LIN {X 0,Y 179.067,Z 302.942,A -85,B 0,C 180,E1 -23619.497,E2 -23619.497} C_VEL
LIN {X 0,Y 181.423,Z 310.34,A -85,B 0,C 180,E1 -23622.061,E2 -23622.061} C_VEL
LIN {X 0,Y 182.867,Z 318.039,A -85,B 0,C 180,E1 -23624.448,E2 -23624.448} C_VEL
LIN {X 0,Y 183.604,Z 326.943,A -85,B 0,C 180,E1 -23627.105,E2 -23627.105} C_VEL
LIN {X 0,Y 183.542,Z 336.442,A -85,B 0,C 180,E1 -23629.98,E2 -23629.98} C_VEL
LIN {X 0,Y 183.368,Z 338.748,A -85,B 0,C 180,E1 -23630.712,E2 -23630.712} C_VEL
LIN {X 0,Y 178.856,Z 348.683,A -85,B 0,C 180,E1 -23633.185,E2 -23633.185} C_VEL
LIN {X 0,Y 173.994,Z 358.418,A -85,B 0,C 180,E1 -23636.262,E2 -23636.262} C_VEL
LIN {X 0,Y 169.557,Z 366.492,A -85,B 0,C 180,E1 -23639.486,E2 -23639.486} C_VEL
LIN {X 0,Y 165.463,Z 373.643,A -85,B 0,C 180,E1 -23643.123,E2 -23643.123} C_VEL
LIN {X 0,Y 162.202,Z 379.606,A -85,B 0,C 180,E1 -23647.048,E2 -23647.048} C_VEL
LIN {X 0,Y 158.721,Z 385.275,A -85,B 0,C 180,E1 -23651.944,E2 -23651.944} C_VEL
LIN {X 0,Y 156.544,Z 389.385,A -85,B 0,C 180,E1 -23657.028,E2 -23657.028} C_VEL
LIN {X 0,Y 155.24,Z 392.068,A -85,B 0,C 180,E1 -23662.194,E2 -23662.194} C_VEL
LIN {X 0,Y 154.776,Z 393.405,A -85,B 0,C 180,E1 -23667.398,E2 -23667.398} C_VEL
LIN {X 0,Y 154.745,Z 393.581,A -85,B 0,C 180,E1 -23670,E2 -23670} C_VEL
LIN {X 0,Y 154.935,Z 392.95,A -85,B 0,C 180,E1 -23675.205,E2 -23675.205} C_VEL
LIN {X 0,Y 155.776,Z 390.989,A -85,B 0,C 180,E1 -23680.397,E2 -23680.397} C_VEL
LIN {X 0,Y 157.497,Z 387.65,A -85,B 0,C 180,E1 -23685.53,E2 -23685.53} C_VEL
LIN {X 0,Y 159.441,Z 384.203,A -85,B 0,C 180,E1 -23689.305,E2 -23689.305} C_VEL
LIN {X 0,Y 162.138,Z 379.816,A -85,B 0,C 180,E1 -23692.962,E2 -23692.962} C_VEL
LIN {X 0,Y 165.058,Z 374.417,A -85,B 0,C 180,E1 -23696.599,E2 -23696.599} C_VEL
LIN {X 0,Y 169.475,Z 366.809,A -85,B 0,C 180,E1 -23700.531,E2 -23700.531} C_VEL
LIN {X 0,Y 173.917,Z 358.8,A -85,B 0,C 180,E1 -23703.755,E2 -23703.755} C_VEL
LIN {X 0,Y 178.733,Z 349.14,A -85,B 0,C 180,E1 -23706.845,E2 -23706.845} C_VEL
LIN {X 0,Y 183.37,Z 339.114,A -85,B 0,C 180,E1 -23709.349,E2 -23709.349} C_VEL
LIN {X 0,Y 183.799,Z 330.673,A -85,B 0,C 180,E1 -23711.941,E2 -23711.941} C_VEL
LIN {X 0,Y 183.309,Z 320.833,A -85,B 0,C 180,E1 -23714.875,E2 -23714.875} C_VEL
LIN {X 0,Y 181.97,Z 312.358,A -85,B 0,C 180,E1 -23717.475,E2 -23717.475} C_VEL
LIN {X 0,Y 179.973,Z 305.35,A -85,B 0,C 180,E1 -23719.831,E2 -23719.831} C_VEL
LIN {X 0,Y 177.108,Z 298.214,A -85,B 0,C 180,E1 -23722.528,E2 -23722.528} C_VEL
LIN {X 0,Y 174.424,Z 292.131,A -85,B 0,C 180,E1 -23724.958,E2 -23724.958} C_VEL
LIN {X 0,Y 171.473,Z 286.759,A -85,B 0,C 180,E1 -23727.456,E2 -23727.456} C_VEL
LIN {X 0,Y 168.98,Z 282.347,A -85,B 0,C 180,E1 -23729.657,E2 -23729.657} C_VEL
LIN {X 0,Y 166.592,Z 279.117,A -85,B 0,C 180,E1 -23731.666,E2 -23731.666} C_VEL
LIN {X 0,Y 165.823,Z 277.609,A -85,B 0,C 180,E1 -23732.439,E2 -23732.439} C_VEL
LIN {X 0,Y 163.535,Z 275.533,A -85,B 0,C 180,E1 -23734.403,E2 -23734.403} C_VEL
LIN {X 0,Y 162.075,Z 272.586,A -85,B 0,C 180,E1 -23736.004,E2 -23736.004} C_VEL
LIN {X 0,Y 158.994,Z 270.202,A -85,B 0,C 180,E1 -23739.121,E2 -23739.121} C_VEL
LIN {X 0,Y 157.602,Z 267.461,A -85,B 0,C 180,E1 -23740.958,E2 -23740.958} C_VEL
LIN {X 0,Y 157.402,Z 266.502,A -85,B 0,C 180,E1 -23741.446,E2 -23741.446} C_VEL
LIN {X 0,Y 157.532,Z 266.485,A -85,B 0,C 180,E1 -23747.111,E2 -23747.111} C_VEL
LIN {X 0,Y 157.691,Z 266.465,A -85,B 0,C 180,E1 -23749.731,E2 -23749.731} C_VEL
LIN {X 0,Y 157.768,Z 266.455,A -85,B 0,C 180,E1 -23752.32,E2 -23752.32} C_VEL
LIN {X 0,Y 158.247,Z 266.395,A -85,B 0,C 180,E1 -23760,E2 -23760} C_VEL
LIN {X 0,Y 157.764,Z 266.456,A -85,B 0,C 180,E1 -23767.68,E2 -23767.68} C_VEL
LIN {X 0,Y 157.635,Z 266.476,A -85,B 0,C 180,E1 -23771.228,E2 -23771.228} C_VEL
LIN {X 0,Y 157.436,Z 266.501,A -85,B 0,C 180,E1 -23775.536,E2 -23775.536} C_VEL
LIN {X 0,Y 157.532,Z 267.283,A -85,B 0,C 180,E1 -23778.666,E2 -23778.666} C_VEL
LIN {X 0,Y 158.727,Z 270.174,A -85,B 0,C 180,E1 -23780.334,E2 -23780.334} C_VEL
LIN {X 0,Y 161.142,Z 273.06,A -85,B 0,C 180,E1 -23782.942,E2 -23782.942} C_VEL
LIN {X 0,Y 162.364,Z 274.144,A -85,B 0,C 180,E1 -23784.111,E2 -23784.111} C_VEL
LIN {X 0,Y 164.013,Z 277.665,A -85,B 0,C 180,E1 -23785.9,E2 -23785.9} C_VEL
LIN {X 0,Y 166.386,Z 280.501,A -85,B 0,C 180,E1 -23787.967,E2 -23787.967} C_VEL
LIN {X 0,Y 168.328,Z 284.343,A -85,B 0,C 180,E1 -23789.809,E2 -23789.809} C_VEL
LIN {X 0,Y 169.782,Z 286.384,A -85,B 0,C 180,E1 -23790.977,E2 -23790.977} C_VEL
LIN {X 0,Y 172.139,Z 290.716,A -85,B 0,C 180,E1 -23793.01,E2 -23793.01} C_VEL
LIN {X 0,Y 176.395,Z 299.815,A -85,B 0,C 180,E1 -23796.701,E2 -23796.701} C_VEL
LIN {X 0,Y 179.977,Z 309.787,A -85,B 0,C 180,E1 -23800.222,E2 -23800.222} C_VEL
LIN {X 0,Y 181.352,Z 315.544,A -85,B 0,C 180,E1 -23802.016,E2 -23802.016} C_VEL
LIN {X 0,Y 182.317,Z 324.212,A -85,B 0,C 180,E1 -23804.451,E2 -23804.451} C_VEL
LIN {X 0,Y 182.511,Z 333.34,A -85,B 0,C 180,E1 -23807.024,E2 -23807.024} C_VEL
LIN {X 0,Y 181.857,Z 342.337,A -85,B 0,C 180,E1 -23809.595,E2 -23809.595} C_VEL
LIN {X 0,Y 181.369,Z 346.338,A -85,B 0,C 180,E1 -23810.804,E2 -23810.804} C_VEL
LIN {X 0,Y 178.739,Z 352.649,A -85,B 0,C 180,E1 -23812.449,E2 -23812.449} C_VEL
LIN {X 0,Y 173.678,Z 362.679,A -85,B 0,C 180,E1 -23815.492,E2 -23815.492} C_VEL
LIN {X 0,Y 169.218,Z 371.013,A -85,B 0,C 180,E1 -23818.724,E2 -23818.724} C_VEL
LIN {X 0,Y 164.754,Z 378.985,A -85,B 0,C 180,E1 -23822.705,E2 -23822.705} C_VEL
LIN {X 0,Y 161.215,Z 385.41,A -85,B 0,C 180,E1 -23826.899,E2 -23826.899} C_VEL
LIN {X 0,Y 158.016,Z 391.107,A -85,B 0,C 180,E1 -23831.86,E2 -23831.86} C_VEL
LIN {X 0,Y 155.897,Z 395.243,A -85,B 0,C 180,E1 -23836.973,E2 -23836.973} C_VEL
LIN {X 0,Y 154.871,Z 397.949,A -85,B 0,C 180,E1 -23842.175,E2 -23842.175} C_VEL
LIN {X 0,Y 154.685,Z 398.789,A -85,B 0,C 180,E1 -23844.786,E2 -23844.786} C_VEL
LIN {X 0,Y 154.744,Z 399.455,A -85,B 0,C 180,E1 -23850,E2 -23850} C_VEL
LIN {X 0,Y 154.683,Z 398.767,A -85,B 0,C 180,E1 -23855.213,E2 -23855.213} C_VEL
LIN {X 0,Y 155.277,Z 396.729,A -85,B 0,C 180,E1 -23860.43,E2 -23860.43} C_VEL
LIN {X 0,Y 156.762,Z 393.297,A -85,B 0,C 180,E1 -23865.604,E2 -23865.604} C_VEL
LIN {X 0,Y 159.448,Z 388.372,A -85,B 0,C 180,E1 -23870.647,E2 -23870.647} C_VEL
LIN {X 0,Y 162.167,Z 383.399,A -85,B 0,C 180,E1 -23874.481,E2 -23874.481} C_VEL
LIN {X 0,Y 165.93,Z 376.75,A -85,B 0,C 180,E1 -23878.457,E2 -23878.457} C_VEL
LIN {X 0,Y 167.766,Z 373.489,A -85,B 0,C 180,E1 -23880.084,E2 -23880.084} C_VEL
LIN {X 0,Y 169.015,Z 370.186,A -85,B 0,C 180,E1 -23881.698,E2 -23881.698} C_VEL
LIN {X 0,Y 169.665,Z 364.547,A -85,B 0,C 180,E1 -23884.452,E2 -23884.452} C_VEL
LIN {X 0,Y 170.538,Z 358.436,A -85,B 0,C 180,E1 -23887.058,E2 -23887.058} C_VEL
LIN {X 0,Y 172.074,Z 354.374,A -85,B 0,C 180,E1 -23888.397,E2 -23888.397} C_VEL
LIN {X 0,Y 174.942,Z 348.416,A -85,B 0,C 180,E1 -23889.999,E2 -23889.999} C_VEL
LIN {X 0,Y 176.332,Z 338.706,A -85,B 0,C 180,E1 -23893.011,E2 -23893.011} C_VEL
LIN {X 0,Y 176.669,Z 328.607,A -85,B 0,C 180,E1 -23896.035,E2 -23896.035} C_VEL
LIN {X 0,Y 176.019,Z 319.46,A -85,B 0,C 180,E1 -23898.793,E2 -23898.793} C_VEL
LIN {X 0,Y 174.653,Z 312.885,A -85,B 0,C 180,E1 -23900.986,E2 -23900.986} C_VEL
LIN {X 0,Y 171.698,Z 304.092,A -85,B 0,C 180,E1 -23904.318,E2 -23904.318} C_VEL
LIN {X 0,Y 168.228,Z 295.98,A -85,B 0,C 180,E1 -23907.815,E2 -23907.815} C_VEL
LIN {X 0,Y 165.717,Z 291.022,A -85,B 0,C 180,E1 -23910.287,E2 -23910.287} C_VEL
LIN {X 0,Y 163.651,Z 287.391,A -85,B 0,C 180,E1 -23912.332,E2 -23912.332} C_VEL
LIN {X 0,Y 163.002,Z 285.935,A -85,B 0,C 180,E1 -23913.082,E2 -23913.082} C_VEL
LIN {X 0,Y 160.702,Z 282.751,A -85,B 0,C 180,E1 -23915.371,E2 -23915.371} C_VEL
LIN {X 0,Y 159.58,Z 280.103,A -85,B 0,C 180,E1 -23916.821,E2 -23916.821} C_VEL
LIN {X 0,Y 156.897,Z 277.104,A -85,B 0,C 180,E1 -23919.849,E2 -23919.849} C_VEL
LIN {X 0,Y 155.347,Z 273.679,A -85,B 0,C 180,E1 -23922.22,E2 -23922.22} C_VEL
LIN {X 0,Y 151.929,Z 270.812,A -85,B 0,C 180,E1 -23927.587,E2 -23927.587} C_VEL
LIN {X 0,Y 150.752,Z 267.956,A -85,B 0,C 180,E1 -23930.694,E2 -23930.694} C_VEL
LIN {X 0,Y 150.654,Z 267.344,A -85,B 0,C 180,E1 -23931.28,E2 -23931.28} C_VEL
LIN {X 0,Y 150.892,Z 267.312,A -85,B 0,C 180,E1 -23937.331,E2 -23937.331} C_VEL
LIN {X 0,Y 151.215,Z 267.273,A -85,B 0,C 180,E1 -23940,E2 -23940} C_VEL
LIN {X 0,Y 150.706,Z 267.338,A -85,B 0,C 180,E1 -23948.042,E2 -23948.042} C_VEL
LIN {X 0,Y 150.671,Z 267.462,A -85,B 0,C 180,E1 -23949.312,E2 -23949.312} C_VEL
LIN {X 0,Y 151.617,Z 270.359,A -85,B 0,C 180,E1 -23952.124,E2 -23952.124} C_VEL
LIN {X 0,Y 153.898,Z 272.667,A -85,B 0,C 180,E1 -23956.243,E2 -23956.243} C_VEL
LIN {X 0,Y 155.476,Z 273.555,A -85,B 0,C 180,E1 -23958.363,E2 -23958.363} C_VEL
LIN {X 0,Y 156.748,Z 276.518,A -85,B 0,C 180,E1 -23960.35,E2 -23960.35} C_VEL
LIN {X 0,Y 159.096,Z 278.658,A -85,B 0,C 180,E1 -23963.021,E2 -23963.021} C_VEL
LIN {X 0,Y 159.656,Z 279.316,A -85,B 0,C 180,E1 -23963.64,E2 -23963.64} C_VEL
LIN {X 0,Y 161.407,Z 282.44,A -85,B 0,C 180,E1 -23965.668,E2 -23965.668} C_VEL
LIN {X 0,Y 163.234,Z 284.363,A -85,B 0,C 180,E1 -23967.397,E2 -23967.397} C_VEL
LIN {X 0,Y 165.077,Z 287.673,A -85,B 0,C 180,E1 -23969.315,E2 -23969.315} C_VEL
LIN {X 0,Y 166.892,Z 290.685,A -85,B 0,C 180,E1 -23971.055,E2 -23971.055} C_VEL
LIN {X 0,Y 168.682,Z 294.057,A -85,B 0,C 180,E1 -23972.795,E2 -23972.795} C_VEL
LIN {X 0,Y 171.593,Z 300.422,A -85,B 0,C 180,E1 -23975.707,E2 -23975.707} C_VEL
LIN {X 0,Y 174.378,Z 307.594,A -85,B 0,C 180,E1 -23978.661,E2 -23978.661} C_VEL
LIN {X 0,Y 176.279,Z 314.277,A -85,B 0,C 180,E1 -23981.134,E2 -23981.134} C_VEL
LIN {X 0,Y 177.396,Z 321.698,A -85,B 0,C 180,E1 -23983.604,E2 -23983.604} C_VEL
LIN {X 0,Y 177.79,Z 330.811,A -85,B 0,C 180,E1 -23986.487,E2 -23986.487} C_VEL
LIN {X 0,Y 177.353,Z 340.066,A -85,B 0,C 180,E1 -23989.516,E2 -23989.516} C_VEL
LIN {X 0,Y 172.297,Z 350.598,A -85,B 0,C 180,E1 -23992.277,E2 -23992.277} C_VEL
LIN {X 0,Y 167.318,Z 360.036,A -85,B 0,C 180,E1 -23995.455,E2 -23995.455} C_VEL
LIN {X 0,Y 162.038,Z 369.033,A -85,B 0,C 180,E1 -23999.361,E2 -23999.361} C_VEL
LIN {X 0,Y 157.689,Z 376.278,A -85,B 0,C 180,E1 -24003.533,E2 -24003.533} C_VEL
LIN {X 0,Y 154.631,Z 381.346,A -85,B 0,C 180,E1 -24007.274,E2 -24007.274} C_VEL
LIN {X 0,Y 151.296,Z 386.595,A -85,B 0,C 180,E1 -24012.426,E2 -24012.426} C_VEL
LIN {X 0,Y 149.628,Z 389.521,A -85,B 0,C 180,E1 -24016.418,E2 -24016.418} C_VEL
LIN {X 0,Y 148.211,Z 392.204,A -85,B 0,C 180,E1 -24021.822,E2 -24021.822} C_VEL
LIN {X 0,Y 147.68,Z 393.54,A -85,B 0,C 180,E1 -24027.273,E2 -24027.273} C_VEL
LIN {X 0,Y 147.631,Z 393.649,A -85,B 0,C 180,E1 -24031.363,E2 -24031.363} C_VEL
LIN {X 0,Y 147.861,Z 393.084,A -85,B 0,C 180,E1 -24035.455,E2 -24035.455} C_VEL
LIN {X 0,Y 148.777,Z 391.124,A -85,B 0,C 180,E1 -24040.892,E2 -24040.892} C_VEL
LIN {X 0,Y 150.649,Z 387.785,A -85,B 0,C 180,E1 -24046.255,E2 -24046.255} C_VEL
LIN {X 0,Y 152.738,Z 384.337,A -85,B 0,C 180,E1 -24050.188,E2 -24050.188} C_VEL
LIN {X 0,Y 155.581,Z 379.951,A -85,B 0,C 180,E1 -24053.989,E2 -24053.989} C_VEL
LIN {X 0,Y 158.893,Z 374.274,A -85,B 0,C 180,E1 -24057.915,E2 -24057.915} C_VEL
LIN {X 0,Y 163.392,Z 366.942,A -85,B 0,C 180,E1 -24061.797,E2 -24061.797} C_VEL
LIN {X 0,Y 168.039,Z 358.933,A -85,B 0,C 180,E1 -24065.105,E2 -24065.105} C_VEL
LIN {X 0,Y 173.103,Z 349.272,A -85,B 0,C 180,E1 -24068.255,E2 -24068.255} C_VEL
LIN {X 0,Y 177.411,Z 340.434,A -85,B 0,C 180,E1 -24070.528,E2 -24070.528} C_VEL
LIN {X 0,Y 177.889,Z 332.538,A -85,B 0,C 180,E1 -24073.106,E2 -24073.106} C_VEL
LIN {X 0,Y 177.721,Z 324.154,A -85,B 0,C 180,E1 -24075.775,E2 -24075.775} C_VEL
LIN {X 0,Y 176.688,Z 316.064,A -85,B 0,C 180,E1 -24078.431,E2 -24078.431} C_VEL
LIN {X 0,Y 175.206,Z 310.11,A -85,B 0,C 180,E1 -24080.573,E2 -24080.573} C_VEL
LIN {X 0,Y 172.379,Z 302.202,A -85,B 0,C 180,E1 -24083.759,E2 -24083.759} C_VEL
LIN {X 0,Y 168.362,Z 293.124,A -85,B 0,C 180,E1 -24087.844,E2 -24087.844} C_VEL
LIN {X 0,Y 165.703,Z 288.288,A -85,B 0,C 180,E1 -24090.458,E2 -24090.458} C_VEL
LIN {X 0,Y 163.476,Z 284.804,A -85,B 0,C 180,E1 -24092.647,E2 -24092.647} C_VEL
LIN {X 0,Y 162.93,Z 283.848,A -85,B 0,C 180,E1 -24093.242,E2 -24093.242} C_VEL
LIN {X 0,Y 160.632,Z 281.334,A -85,B 0,C 180,E1 -24095.487,E2 -24095.487} C_VEL
LIN {X 0,Y 159.396,Z 278.805,A -85,B 0,C 180,E1 -24097.049,E2 -24097.049} C_VEL
LIN {X 0,Y 157.027,Z 276.836,A -85,B 0,C 180,E1 -24099.705,E2 -24099.705} C_VEL
LIN {X 0,Y 155.571,Z 273.871,A -85,B 0,C 180,E1 -24101.906,E2 -24101.906} C_VEL
LIN {X 0,Y 155.406,Z 273.314,A -85,B 0,C 180,E1 -24102.226,E2 -24102.226} C_VEL
LIN {X 0,Y 152.481,Z 271.504,A -85,B 0,C 180,E1 -24106.676,E2 -24106.676} C_VEL
LIN {X 0,Y 150.953,Z 268.682,A -85,B 0,C 180,E1 -24110.453,E2 -24110.453} C_VEL
LIN {X 0,Y 150.692,Z 267.336,A -85,B 0,C 180,E1 -24111.788,E2 -24111.788} C_VEL
LIN {X 0,Y 151.209,Z 267.272,A -85,B 0,C 180,E1 -24120,E2 -24120} C_VEL
LIN {X 0,Y 150.719,Z 267.523,A -85,B 0,C 180,E1 -24128.294,E2 -24128.294} C_VEL
LIN {X 0,Y 151.32,Z 269.624,A -85,B 0,C 180,E1 -24130.368,E2 -24130.368} C_VEL
LIN {X 0,Y 153.209,Z 272.203,A -85,B 0,C 180,E1 -24134.274,E2 -24134.274} C_VEL
LIN {X 0,Y 155.638,Z 274.025,A -85,B 0,C 180,E1 -24137.831,E2 -24137.831} C_VEL
LIN {X 0,Y 157.461,Z 277.866,A -85,B 0,C 180,E1 -24140.544,E2 -24140.544} C_VEL
LIN {X 0,Y 159.847,Z 280.493,A -85,B 0,C 180,E1 -24143.224,E2 -24143.224} C_VEL
LIN {X 0,Y 161.591,Z 284.192,A -85,B 0,C 180,E1 -24145.349,E2 -24145.349} C_VEL
LIN {X 0,Y 163.459,Z 286.72,A -85,B 0,C 180,E1 -24147.182,E2 -24147.182} C_VEL
LIN {X 0,Y 165.243,Z 290.402,A -85,B 0,C 180,E1 -24149.107,E2 -24149.107} C_VEL
LIN {X 0,Y 166.06,Z 291.49,A -85,B 0,C 180,E1 -24149.82,E2 -24149.82} C_VEL
LIN {X 0,Y 168.947,Z 297.6,A -85,B 0,C 180,E1 -24152.737,E2 -24152.737} C_VEL
LIN {X 0,Y 172.405,Z 305.804,A -85,B 0,C 180,E1 -24156.234,E2 -24156.234} C_VEL
LIN {X 0,Y 174.848,Z 313.347,A -85,B 0,C 180,E1 -24159.08,E2 -24159.08} C_VEL
LIN {X 0,Y 176.143,Z 319.606,A -85,B 0,C 180,E1 -24161.172,E2 -24161.172} C_VEL
LIN {X 0,Y 176.759,Z 328.96,A -85,B 0,C 180,E1 -24163.984,E2 -24163.984} C_VEL
LIN {X 0,Y 176.519,Z 337.676,A -85,B 0,C 180,E1 -24166.601,E2 -24166.601} C_VEL
LIN {X 0,Y 175.31,Z 347.396,A -85,B 0,C 180,E1 -24169.613,E2 -24169.613} C_VEL
LIN {X 0,Y 174.02,Z 350.627,A -85,B 0,C 180,E1 -24170.499,E2 -24170.499} C_VEL
LIN {X 0,Y 168.732,Z 361.032,A -85,B 0,C 180,E1 -24173.591,E2 -24173.591} C_VEL
LIN {X 0,Y 163.915,Z 369.618,A -85,B 0,C 180,E1 -24176.861,E2 -24176.861} C_VEL
LIN {X 0,Y 159.05,Z 377.839,A -85,B 0,C 180,E1 -24180.918,E2 -24180.918} C_VEL
LIN {X 0,Y 155.539,Z 383.693,A -85,B 0,C 180,E1 -24184.648,E2 -24184.648} C_VEL
LIN {X 0,Y 152.791,Z 388.328,A -85,B 0,C 180,E1 -24188.409,E2 -24188.409} C_VEL
LIN {X 0,Y 149.896,Z 393.225,A -85,B 0,C 180,E1 -24193.661,E2 -24193.661} C_VEL
LIN {X 0,Y 148.272,Z 396.635,A -85,B 0,C 180,E1 -24199.07,E2 -24199.07} C_VEL
LIN {X 0,Y 147.612,Z 398.654,A -85,B 0,C 180,E1 -24204.536,E2 -24204.536} C_VEL
LIN {X 0,Y 147.656,Z 399.32,A -85,B 0,C 180,E1 -24210,E2 -24210} C_VEL
LIN {X 0,Y 147.61,Z 398.632,A -85,B 0,C 180,E1 -24215.464,E2 -24215.464} C_VEL
LIN {X 0,Y 148.271,Z 396.594,A -85,B 0,C 180,E1 -24220.929,E2 -24220.929} C_VEL
LIN {X 0,Y 149.892,Z 393.16,A -85,B 0,C 180,E1 -24226.339,E2 -24226.339} C_VEL
LIN {X 0,Y 152.778,Z 388.235,A -85,B 0,C 180,E1 -24231.593,E2 -24231.593} C_VEL
LIN {X 0,Y 156.652,Z 381.67,A -85,B 0,C 180,E1 -24236.656,E2 -24236.656} C_VEL
LIN {X 0,Y 161.019,Z 374.371,A -85,B 0,C 180,E1 -24240.854,E2 -24240.854} C_VEL
LIN {X 0,Y 166.195,Z 365.331,A -85,B 0,C 180,E1 -24244.812,E2 -24244.812} C_VEL
LIN {X 0,Y 171.334,Z 355.855,A -85,B 0,C 180,E1 -24247.973,E2 -24247.973} C_VEL
LIN {X 0,Y 172.074,Z 354.374,A -85,B 0,C 180,E1 -24248.397,E2 -24248.397} C_VEL
LIN {X 0,Y 173.06,Z 351.66,A -85,B 0,C 180,E1 -24249.261,E2 -24249.261} C_VEL
LIN {X 0,Y 173.329,Z 347.715,A -85,B 0,C 180,E1 -24250.724,E2 -24250.724} C_VEL
LIN {X 0,Y 172.71,Z 344.045,A -85,B 0,C 180,E1 -24252.275,E2 -24252.275} C_VEL
LIN {X 0,Y 171.017,Z 336.395,A -85,B 0,C 180,E1 -24255.458,E2 -24255.458} C_VEL
LIN {X 0,Y 170.946,Z 333.508,A -85,B 0,C 180,E1 -24256.433,E2 -24256.433} C_VEL
LIN {X 0,Y 170.857,Z 324.847,A -85,B 0,C 180,E1 -24259.204,E2 -24259.204} C_VEL
LIN {X 0,Y 169.871,Z 317.824,A -85,B 0,C 180,E1 -24261.641,E2 -24261.641} C_VEL
LIN {X 0,Y 167.569,Z 309.915,A -85,B 0,C 180,E1 -24264.809,E2 -24264.809} C_VEL
LIN {X 0,Y 164.492,Z 301.734,A -85,B 0,C 180,E1 -24268.513,E2 -24268.513} C_VEL
LIN {X 0,Y 162.458,Z 297.122,A -85,B 0,C 180,E1 -24270.878,E2 -24270.878} C_VEL
LIN {X 0,Y 159.428,Z 291.4,A -85,B 0,C 180,E1 -24274.37,E2 -24274.37} C_VEL
LIN {X 0,Y 157.388,Z 287.639,A -85,B 0,C 180,E1 -24276.914,E2 -24276.914} C_VEL
LIN {X 0,Y 156.806,Z 286.281,A -85,B 0,C 180,E1 -24277.78,E2 -24277.78} C_VEL
LIN {X 0,Y 154.507,Z 283.311,A -85,B 0,C 180,E1 -24280.75,E2 -24280.75} C_VEL
LIN {X 0,Y 153.427,Z 280.414,A -85,B 0,C 180,E1 -24282.764,E2 -24282.764} C_VEL
LIN {X 0,Y 150.236,Z 277.448,A -85,B 0,C 180,E1 -24288.331,E2 -24288.331} C_VEL
LIN {X 0,Y 149.201,Z 274.279,A -85,B 0,C 180,E1 -24291.876,E2 -24291.876} C_VEL
LIN {X 0,Y 147.773,Z 273.479,A -85,B 0,C 180,E1 -24300,E2 -24300} C_VEL
LIN {X 0,Y 149.213,Z 274.312,A -85,B 0,C 180,E1 -24308.635,E2 -24308.635} C_VEL
LIN {X 0,Y 150.133,Z 277.31,A -85,B 0,C 180,E1 -24311.912,E2 -24311.912} C_VEL
LIN {X 0,Y 152.264,Z 279.562,A -85,B 0,C 180,E1 -24316.078,E2 -24316.078} C_VEL
LIN {X 0,Y 153.329,Z 280.245,A -85,B 0,C 180,E1 -24317.636,E2 -24317.636} C_VEL
LIN {X 0,Y 154.634,Z 283.227,A -85,B 0,C 180,E1 -24319.93,E2 -24319.93} C_VEL
LIN {X 0,Y 156.999,Z 285.641,A -85,B 0,C 180,E1 -24322.886,E2 -24322.886} C_VEL
LIN {X 0,Y 158.503,Z 288.594,A -85,B 0,C 180,E1 -24324.912,E2 -24324.912} C_VEL
LIN {X 0,Y 159.669,Z 289.817,A -85,B 0,C 180,E1 -24326.114,E2 -24326.114} C_VEL
LIN {X 0,Y 162.989,Z 295.615,A -85,B 0,C 180,E1 -24329.87,E2 -24329.87} C_VEL
LIN {X 0,Y 166.061,Z 302.275,A -85,B 0,C 180,E1 -24333.38,E2 -24333.38} C_VEL
LIN {X 0,Y 169.043,Z 310.375,A -85,B 0,C 180,E1 -24337.075,E2 -24337.075} C_VEL
LIN {X 0,Y 171.126,Z 318.459,A -85,B 0,C 180,E1 -24340.304,E2 -24340.304} C_VEL
LIN {X 0,Y 171.991,Z 326.656,A -85,B 0,C 180,E1 -24343.193,E2 -24343.193} C_VEL
LIN {X 0,Y 171.835,Z 336.017,A -85,B 0,C 180,E1 -24346.356,E2 -24346.356} C_VEL
LIN {X 0,Y 171.376,Z 341.47,A -85,B 0,C 180,E1 -24348.257,E2 -24348.257} C_VEL
LIN {X 0,Y 165.839,Z 352.438,A -85,B 0,C 180,E1 -24351.312,E2 -24351.312} C_VEL
LIN {X 0,Y 160.684,Z 361.565,A -85,B 0,C 180,E1 -24354.583,E2 -24354.583} C_VEL
LIN {X 0,Y 155.229,Z 370.282,A -85,B 0,C 180,E1 -24358.624,E2 -24358.624} C_VEL
LIN {X 0,Y 151.343,Z 376.414,A -85,B 0,C 180,E1 -24362.33,E2 -24362.33} C_VEL
LIN {X 0,Y 148.092,Z 381.482,A -85,B 0,C 180,E1 -24366.21,E2 -24366.21} C_VEL
LIN {X 0,Y 144.512,Z 386.731,A -85,B 0,C 180,E1 -24371.572,E2 -24371.572} C_VEL
LIN {X 0,Y 142.708,Z 389.657,A -85,B 0,C 180,E1 -24375.745,E2 -24375.745} C_VEL
LIN {X 0,Y 141.165,Z 392.339,A -85,B 0,C 180,E1 -24381.411,E2 -24381.411} C_VEL
LIN {X 0,Y 140.594,Z 393.675,A -85,B 0,C 180,E1 -24387.135,E2 -24387.135} C_VEL
LIN {X 0,Y 140.561,Z 393.85,A -85,B 0,C 180,E1 -24390,E2 -24390} C_VEL
LIN {X 0,Y 140.799,Z 393.219,A -85,B 0,C 180,E1 -24395.73,E2 -24395.73} C_VEL
LIN {X 0,Y 141.802,Z 391.258,A -85,B 0,C 180,E1 -24401.435,E2 -24401.435} C_VEL
LIN {X 0,Y 143.81,Z 387.919,A -85,B 0,C 180,E1 -24407.051,E2 -24407.051} C_VEL
LIN {X 0,Y 146.077,Z 384.471,A -85,B 0,C 180,E1 -24411.152,E2 -24411.152} C_VEL
LIN {X 0,Y 149.064,Z 380.085,A -85,B 0,C 180,E1 -24415.108,E2 -24415.108} C_VEL
LIN {X 0,Y 152.837,Z 374.089,A -85,B 0,C 180,E1 -24419.365,E2 -24419.365} C_VEL
LIN {X 0,Y 158.174,Z 365.848,A -85,B 0,C 180,E1 -24423.739,E2 -24423.739} C_VEL
LIN {X 0,Y 163.13,Z 357.585,A -85,B 0,C 180,E1 -24427.096,E2 -24427.096} C_VEL
LIN {X 0,Y 168.517,Z 347.628,A -85,B 0,C 180,E1 -24430.273,E2 -24430.273} C_VEL
LIN {X 0,Y 171.488,Z 341.782,A -85,B 0,C 180,E1 -24431.788,E2 -24431.788} C_VEL
LIN {X 0,Y 172.12,Z 332.707,A -85,B 0,C 180,E1 -24434.924,E2 -24434.924} C_VEL
LIN {X 0,Y 171.903,Z 323.637,A -85,B 0,C 180,E1 -24438.014,E2 -24438.014} C_VEL
LIN {X 0,Y 170.938,Z 317.042,A -85,B 0,C 180,E1 -24440.411,E2 -24440.411} C_VEL
LIN {X 0,Y 168.729,Z 309.394,A -85,B 0,C 180,E1 -24443.59,E2 -24443.59} C_VEL
LIN {X 0,Y 165.721,Z 301.506,A -85,B 0,C 180,E1 -24447.269,E2 -24447.269} C_VEL
LIN {X 0,Y 164.145,Z 297.962,A -85,B 0,C 180,E1 -24449.083,E2 -24449.083} C_VEL
LIN {X 0,Y 162.622,Z 294.578,A -85,B 0,C 180,E1 -24450.909,E2 -24450.909} C_VEL
LIN {X 0,Y 159.942,Z 290.097,A -85,B 0,C 180,E1 -24453.934,E2 -24453.934} C_VEL
LIN {X 0,Y 157.649,Z 287.113,A -85,B 0,C 180,E1 -24456.519,E2 -24456.519} C_VEL
LIN {X 0,Y 156.934,Z 285.349,A -85,B 0,C 180,E1 -24457.625,E2 -24457.625} C_VEL
LIN {X 0,Y 154.693,Z 283.245,A -85,B 0,C 180,E1 -24460.427,E2 -24460.427} C_VEL
LIN {X 0,Y 153.256,Z 280.015,A -85,B 0,C 180,E1 -24463.001,E2 -24463.001} C_VEL
LIN {X 0,Y 150.609,Z 278.032,A -85,B 0,C 180,E1 -24467.586,E2 -24467.586} C_VEL
LIN {X 0,Y 149.326,Z 274.871,A -85,B 0,C 180,E1 -24471.73,E2 -24471.73} C_VEL
LIN {X 0,Y 149.152,Z 274.273,A -85,B 0,C 180,E1 -24472.555,E2 -24472.555} C_VEL
LIN {X 0,Y 148.078,Z 273.648,A -85,B 0,C 180,E1 -24480,E2 -24480} C_VEL
LIN {X 0,Y 149.308,Z 274.423,A -85,B 0,C 180,E1 -24487.607,E2 -24487.607} C_VEL
LIN {X 0,Y 150.395,Z 277.626,A -85,B 0,C 180,E1 -24491.435,E2 -24491.435} C_VEL
LIN {X 0,Y 153.566,Z 280.712,A -85,B 0,C 180,E1 -24497.113,E2 -24497.113} C_VEL
LIN {X 0,Y 155.445,Z 284.749,A -85,B 0,C 180,E1 -24500.252,E2 -24500.252} C_VEL
LIN {X 0,Y 157.183,Z 286.833,A -85,B 0,C 180,E1 -24502.423,E2 -24502.423} C_VEL
LIN {X 0,Y 158.929,Z 290.681,A -85,B 0,C 180,E1 -24504.841,E2 -24504.841} C_VEL
LIN {X 0,Y 160.077,Z 292.12,A -85,B 0,C 180,E1 -24506.042,E2 -24506.042} C_VEL
LIN {X 0,Y 162.034,Z 296.489,A -85,B 0,C 180,E1 -24508.497,E2 -24508.497} C_VEL
LIN {X 0,Y 164.531,Z 301.686,A -85,B 0,C 180,E1 -24511.316,E2 -24511.316} C_VEL
LIN {X 0,Y 167.86,Z 310.54,A -85,B 0,C 180,E1 -24515.337,E2 -24515.337} C_VEL
LIN {X 0,Y 169.991,Z 318.018,A -85,B 0,C 180,E1 -24518.327,E2 -24518.327} C_VEL
LIN {X 0,Y 170.877,Z 323.847,A -85,B 0,C 180,E1 -24520.374,E2 -24520.374} C_VEL
LIN {X 0,Y 171.063,Z 332.96,A -85,B 0,C 180,E1 -24523.311,E2 -24523.311} C_VEL
LIN {X 0,Y 170.35,Z 342.245,A -85,B 0,C 180,E1 -24526.288,E2 -24526.288} C_VEL
LIN {X 0,Y 169.288,Z 348.534,A -85,B 0,C 180,E1 -24528.375,E2 -24528.375} C_VEL
LIN {X 0,Y 167.55,Z 352.574,A -85,B 0,C 180,E1 -24529.53,E2 -24529.53} C_VEL
LIN {X 0,Y 162.142,Z 362.413,A -85,B 0,C 180,E1 -24532.639,E2 -24532.639} C_VEL
LIN {X 0,Y 157.201,Z 370.746,A -85,B 0,C 180,E1 -24536.024,E2 -24536.024} C_VEL
LIN {X 0,Y 152.185,Z 378.717,A -85,B 0,C 180,E1 -24540.235,E2 -24540.235} C_VEL
LIN {X 0,Y 148.135,Z 385.14,A -85,B 0,C 180,E1 -24544.723,E2 -24544.723} C_VEL
LIN {X 0,Y 144.511,Z 390.837,A -85,B 0,C 180,E1 -24550.096,E2 -24550.096} C_VEL
LIN {X 0,Y 142.02,Z 394.974,A -85,B 0,C 180,E1 -24555.674,E2 -24555.674} C_VEL
LIN {X 0,Y 140.772,Z 397.68,A -85,B 0,C 180,E1 -24561.386,E2 -24561.386} C_VEL
LIN {X 0,Y 140.533,Z 398.519,A -85,B 0,C 180,E1 -24564.259,E2 -24564.259} C_VEL
LIN {X 0,Y 140.56,Z 399.186,A -85,B 0,C 180,E1 -24570,E2 -24570} C_VEL
LIN {X 0,Y 140.532,Z 398.496,A -85,B 0,C 180,E1 -24575.74,E2 -24575.74} C_VEL
LIN {X 0,Y 141.258,Z 396.457,A -85,B 0,C 180,E1 -24581.479,E2 -24581.479} C_VEL
LIN {X 0,Y 143.051,Z 393.024,A -85,B 0,C 180,E1 -24587.144,E2 -24587.144} C_VEL
LIN {X 0,Y 146.159,Z 388.099,A -85,B 0,C 180,E1 -24592.624,E2 -24592.624} C_VEL
LIN {X 0,Y 149.275,Z 383.159,A -85,B 0,C 180,E1 -24596.728,E2 -24596.728} C_VEL
LIN {X 0,Y 153.514,Z 376.475,A -85,B 0,C 180,E1 -24601,E2 -24601} C_VEL
LIN {X 0,Y 158.732,Z 367.946,A -85,B 0,C 180,E1 -24605.141,E2 -24605.141} C_VEL
LIN {X 0,Y 163.919,Z 359.051,A -85,B 0,C 180,E1 -24608.439,E2 -24608.439} C_VEL
LIN {X 0,Y 168.698,Z 350.022,A -85,B 0,C 180,E1 -24611.092,E2 -24611.092} C_VEL
LIN {X 0,Y 169.923,Z 344.11,A -85,B 0,C 180,E1 -24613.034,E2 -24613.034} C_VEL
LIN {X 0,Y 170.809,Z 336.133,A -85,B 0,C 180,E1 -24615.616,E2 -24615.616} C_VEL
LIN {X 0,Y 170.946,Z 333.508,A -85,B 0,C 180,E1 -24616.433,E2 -24616.433} C_VEL
LIN {X 0,Y 170.808,Z 330.777,A -85,B 0,C 180,E1 -24617.38,E2 -24617.38} C_VEL
LIN {X 0,Y 170.131,Z 328.361,A -85,B 0,C 180,E1 -24618.403,E2 -24618.403} C_VEL
LIN {X 0,Y 167.929,Z 324.217,A -85,B 0,C 180,E1 -24620.584,E2 -24620.584} C_VEL
LIN {X 0,Y 164.205,Z 318.223,A -85,B 0,C 180,E1 -24624.035,E2 -24624.035} C_VEL
LIN {X 0,Y 163.342,Z 315.872,A -85,B 0,C 180,E1 -24625.156,E2 -24625.156} C_VEL
LIN {X 0,Y 160.654,Z 307.629,A -85,B 0,C 180,E1 -24629.085,E2 -24629.085} C_VEL
LIN {X 0,Y 158.324,Z 301.993,A -85,B 0,C 180,E1 -24632.22,E2 -24632.22} C_VEL
LIN {X 0,Y 156.551,Z 297.822,A -85,B 0,C 180,E1 -24634.756,E2 -24634.756} C_VEL
LIN {X 0,Y 154.687,Z 294.464,A -85,B 0,C 180,E1 -24637.283,E2 -24637.283} C_VEL
LIN {X 0,Y 153.959,Z 292.502,A -85,B 0,C 180,E1 -24638.581,E2 -24638.581} C_VEL
LIN {X 0,Y 151.827,Z 289.282,A -85,B 0,C 180,E1 -24641.793,E2 -24641.793} C_VEL
LIN {X 0,Y 151.118,Z 287.004,A -85,B 0,C 180,E1 -24643.45,E2 -24643.45} C_VEL
LIN {X 0,Y 148.276,Z 284.016,A -85,B 0,C 180,E1 -24649.071,E2 -24649.071} C_VEL
LIN {X 0,Y 147.501,Z 281.157,A -85,B 0,C 180,E1 -24652.471,E2 -24652.471} C_VEL
LIN {X 0,Y 146.31,Z 280.423,A -85,B 0,C 180,E1 -24660,E2 -24660} C_VEL
LIN {X 0,Y 147.508,Z 281.308,A -85,B 0,C 180,E1 -24668.218,E2 -24668.218} C_VEL
LIN {X 0,Y 148.285,Z 284.173,A -85,B 0,C 180,E1 -24671.621,E2 -24671.621} C_VEL
LIN {X 0,Y 150.536,Z 286.477,A -85,B 0,C 180,E1 -24676.268,E2 -24676.268} C_VEL
LIN {X 0,Y 151.036,Z 287.135,A -85,B 0,C 180,E1 -24677.169,E2 -24677.169} C_VEL
LIN {X 0,Y 151.859,Z 289.247,A -85,B 0,C 180,E1 -24678.903,E2 -24678.903} C_VEL
LIN {X 0,Y 153.608,Z 291.353,A -85,B 0,C 180,E1 -24681.471,E2 -24681.471} C_VEL
LIN {X 0,Y 156.361,Z 295.754,A -85,B 0,C 180,E1 -24685.278,E2 -24685.278} C_VEL
LIN {X 0,Y 159.245,Z 301.173,A -85,B 0,C 180,E1 -24689.043,E2 -24689.043} C_VEL
LIN {X 0,Y 162.045,Z 308.012,A -85,B 0,C 180,E1 -24692.829,E2 -24692.829} C_VEL
LIN {X 0,Y 164.574,Z 316.149,A -85,B 0,C 180,E1 -24696.717,E2 -24696.717} C_VEL
LIN {X 0,Y 165.928,Z 322.553,A -85,B 0,C 180,E1 -24699.445,E2 -24699.445} C_VEL
LIN {X 0,Y 166.371,Z 329.317,A -85,B 0,C 180,E1 -24701.986,E2 -24701.986} C_VEL
LIN {X 0,Y 166.085,Z 337.106,A -85,B 0,C 180,E1 -24704.794,E2 -24704.794} C_VEL
LIN {X 0,Y 165.259,Z 343.463,A -85,B 0,C 180,E1 -24707.123,E2 -24707.123} C_VEL
LIN {X 0,Y 159.416,Z 354.197,A -85,B 0,C 180,E1 -24710.265,E2 -24710.265} C_VEL
LIN {X 0,Y 154.107,Z 363.051,A -85,B 0,C 180,E1 -24713.64,E2 -24713.64} C_VEL
LIN {X 0,Y 148.428,Z 371.53,A -85,B 0,C 180,E1 -24717.813,E2 -24717.813} C_VEL
LIN {X 0,Y 143.835,Z 378.35,A -85,B 0,C 180,E1 -24722.343,E2 -24722.343} C_VEL
LIN {X 0,Y 140.516,Z 383.053,A -85,B 0,C 180,E1 -24726.414,E2 -24726.414} C_VEL
LIN {X 0,Y 137.771,Z 386.867,A -85,B 0,C 180,E1 -24730.636,E2 -24730.636} C_VEL
LIN {X 0,Y 135.82,Z 389.793,A -85,B 0,C 180,E1 -24735.006,E2 -24735.006} C_VEL
LIN {X 0,Y 134.134,Z 392.475,A -85,B 0,C 180,E1 -24740.957,E2 -24740.957} C_VEL
LIN {X 0,Y 133.519,Z 393.81,A -85,B 0,C 180,E1 -24746.983,E2 -24746.983} C_VEL
LIN {X 0,Y 133.475,Z 393.985,A -85,B 0,C 180,E1 -24750,E2 -24750} C_VEL
LIN {X 0,Y 133.731,Z 393.353,A -85,B 0,C 180,E1 -24756.034,E2 -24756.034} C_VEL
LIN {X 0,Y 134.827,Z 391.393,A -85,B 0,C 180,E1 -24762.035,E2 -24762.035} C_VEL
LIN {X 0,Y 137.013,Z 388.054,A -85,B 0,C 180,E1 -24767.925,E2 -24767.925} C_VEL
LIN {X 0,Y 139.465,Z 384.605,A -85,B 0,C 180,E1 -24772.207,E2 -24772.207} C_VEL
LIN {X 0,Y 142.612,Z 380.22,A -85,B 0,C 180,E1 -24776.329,E2 -24776.329} C_VEL
LIN {X 0,Y 146.916,Z 373.878,A -85,B 0,C 180,E1 -24780.947,E2 -24780.947} C_VEL
LIN {X 0,Y 152.312,Z 365.981,A -85,B 0,C 180,E1 -24785.225,E2 -24785.225} C_VEL
LIN {X 0,Y 157.514,Z 357.717,A -85,B 0,C 180,E1 -24788.657,E2 -24788.657} C_VEL
LIN {X 0,Y 163.17,Z 347.759,A -85,B 0,C 180,E1 -24791.883,E2 -24791.883} C_VEL
LIN {X 0,Y 165.574,Z 343.094,A -85,B 0,C 180,E1 -24793.141,E2 -24793.141} C_VEL
LIN {X 0,Y 166.394,Z 334.354,A -85,B 0,C 180,E1 -24796.356,E2 -24796.356} C_VEL
LIN {X 0,Y 166.423,Z 326.815,A -85,B 0,C 180,E1 -24799.115,E2 -24799.115} C_VEL
LIN {X 0,Y 165.477,Z 319.613,A -85,B 0,C 180,E1 -24801.987,E2 -24801.987} C_VEL
LIN {X 0,Y 163.551,Z 312.47,A -85,B 0,C 180,E1 -24805.214,E2 -24805.214} C_VEL
LIN {X 0,Y 161.037,Z 305.378,A -85,B 0,C 180,E1 -24808.82,E2 -24808.82} C_VEL
LIN {X 0,Y 158.809,Z 300.046,A -85,B 0,C 180,E1 -24811.891,E2 -24811.891} C_VEL
LIN {X 0,Y 156.63,Z 296.029,A -85,B 0,C 180,E1 -24814.769,E2 -24814.769} C_VEL
LIN {X 0,Y 154.688,Z 293.204,A -85,B 0,C 180,E1 -24817.283,E2 -24817.283} C_VEL
LIN {X 0,Y 153.902,Z 291.558,A -85,B 0,C 180,E1 -24818.572,E2 -24818.572} C_VEL
LIN {X 0,Y 151.596,Z 288.53,A -85,B 0,C 180,E1 -24822.113,E2 -24822.113} C_VEL
LIN {X 0,Y 150.844,Z 286.661,A -85,B 0,C 180,E1 -24823.767,E2 -24823.767} C_VEL
LIN {X 0,Y 148.425,Z 284.337,A -85,B 0,C 180,E1 -24828.736,E2 -24828.736} C_VEL
LIN {X 0,Y 147.567,Z 281.241,A -85,B 0,C 180,E1 -24832.71,E2 -24832.71} C_VEL
LIN {X 0,Y 146.607,Z 280.598,A -85,B 0,C 180,E1 -24840,E2 -24840} C_VEL
LIN {X 0,Y 147.649,Z 281.398,A -85,B 0,C 180,E1 -24847.178,E2 -24847.178} C_VEL
LIN {X 0,Y 148.763,Z 284.748,A -85,B 0,C 180,E1 -24851.583,E2 -24851.583} C_VEL
LIN {X 0,Y 151.235,Z 287.186,A -85,B 0,C 180,E1 -24856.363,E2 -24856.363} C_VEL
LIN {X 0,Y 152.905,Z 291.155,A -85,B 0,C 180,E1 -24859.64,E2 -24859.64} C_VEL
LIN {X 0,Y 154.179,Z 292.681,A -85,B 0,C 180,E1 -24861.387,E2 -24861.387} C_VEL
LIN {X 0,Y 155.721,Z 296.555,A -85,B 0,C 180,E1 -24863.965,E2 -24863.965} C_VEL
LIN {X 0,Y 156.752,Z 298.021,A -85,B 0,C 180,E1 -24865.21,E2 -24865.21} C_VEL
LIN {X 0,Y 159.429,Z 304.443,A -85,B 0,C 180,E1 -24869.006,E2 -24869.006} C_VEL
LIN {X 0,Y 162.156,Z 311.79,A -85,B 0,C 180,E1 -24872.804,E2 -24872.804} C_VEL
LIN {X 0,Y 164.181,Z 319.004,A -85,B 0,C 180,E1 -24876.058,E2 -24876.058} C_VEL
LIN {X 0,Y 165.319,Z 324.711,A -85,B 0,C 180,E1 -24878.391,E2 -24878.391} C_VEL
LIN {X 0,Y 165.491,Z 332.64,A -85,B 0,C 180,E1 -24881.165,E2 -24881.165} C_VEL
LIN {X 0,Y 164.953,Z 340.46,A -85,B 0,C 180,E1 -24883.827,E2 -24883.827} C_VEL
LIN {X 0,Y 163.388,Z 349.511,A -85,B 0,C 180,E1 -24886.99,E2 -24886.99} C_VEL
LIN {X 0,Y 161.89,Z 352.98,A -85,B 0,C 180,E1 -24888.051,E2 -24888.051} C_VEL
LIN {X 0,Y 156.538,Z 362.28,A -85,B 0,C 180,E1 -24891.056,E2 -24891.056} C_VEL
LIN {X 0,Y 151.342,Z 370.613,A -85,B 0,C 180,E1 -24894.516,E2 -24894.516} C_VEL
LIN {X 0,Y 146.014,Z 378.583,A -85,B 0,C 180,E1 -24898.84,E2 -24898.84} C_VEL
LIN {X 0,Y 141.674,Z 385.005,A -85,B 0,C 180,E1 -24903.483,E2 -24903.483} C_VEL
LIN {X 0,Y 137.825,Z 390.703,A -85,B 0,C 180,E1 -24909.087,E2 -24909.087} C_VEL
LIN {X 0,Y 135.116,Z 394.839,A -85,B 0,C 180,E1 -24914.925,E2 -24914.925} C_VEL
LIN {X 0,Y 133.726,Z 397.545,A -85,B 0,C 180,E1 -24920.928,E2 -24920.928} C_VEL
LIN {X 0,Y 133.449,Z 398.384,A -85,B 0,C 180,E1 -24923.954,E2 -24923.954} C_VEL
LIN {X 0,Y 133.456,Z 399.051,A -85,B 0,C 180,E1 -24930,E2 -24930} C_VEL
LIN {X 0,Y 133.448,Z 398.361,A -85,B 0,C 180,E1 -24936.046,E2 -24936.046} C_VEL
LIN {X 0,Y 134.271,Z 396.321,A -85,B 0,C 180,E1 -24942.085,E2 -24942.085} C_VEL
LIN {X 0,Y 136.25,Z 392.888,A -85,B 0,C 180,E1 -24948.028,E2 -24948.028} C_VEL
LIN {X 0,Y 139.594,Z 387.962,A -85,B 0,C 180,E1 -24953.751,E2 -24953.751} C_VEL
LIN {X 0,Y 142.806,Z 383.216,A -85,B 0,C 180,E1 -24957.872,E2 -24957.872} C_VEL
LIN {X 0,Y 147.446,Z 376.338,A -85,B 0,C 180,E1 -24962.427,E2 -24962.427} C_VEL
LIN {X 0,Y 152.943,Z 367.808,A -85,B 0,C 180,E1 -24966.682,E2 -24966.682} C_VEL
LIN {X 0,Y 158.408,Z 358.913,A -85,B 0,C 180,E1 -24970.039,E2 -24970.039} C_VEL
LIN {X 0,Y 162.786,Z 351.036,A -85,B 0,C 180,E1 -24972.437,E2 -24972.437} C_VEL
LIN {X 0,Y 164.341,Z 343.959,A -85,B 0,C 180,E1 -24974.879,E2 -24974.879} C_VEL
LIN {X 0,Y 165.373,Z 333.727,A -85,B 0,C 180,E1 -24978.369,E2 -24978.369} C_VEL
LIN {X 0,Y 165.316,Z 325.941,A -85,B 0,C 180,E1 -24981.057,E2 -24981.057} C_VEL
LIN {X 0,Y 164.44,Z 320.322,A -85,B 0,C 180,E1 -24983.249,E2 -24983.249} C_VEL
LIN {X 0,Y 163.342,Z 315.872,A -85,B 0,C 180,E1 -24985.156,E2 -24985.156} C_VEL
LIN {X 0,Y 161.869,Z 312.825,A -85,B 0,C 180,E1 -24986.855,E2 -24986.855} C_VEL
LIN {X 0,Y 159.802,Z 310.704,A -85,B 0,C 180,E1 -24988.693,E2 -24988.693} C_VEL
LIN {X 0,Y 155.378,Z 307.374,A -85,B 0,C 180,E1 -24992.594,E2 -24992.594} C_VEL
LIN {X 0,Y 153.673,Z 305.15,A -85,B 0,C 180,E1 -24994.572,E2 -24994.572} C_VEL
LIN {X 0,Y 153.262,Z 304.202,A -85,B 0,C 180,E1 -24995.214,E2 -24995.214} C_VEL
LIN {X 0,Y 150.795,Z 298.454,A -85,B 0,C 180,E1 -24999.541,E2 -24999.541} C_VEL
LIN {X 0,Y 149.246,Z 295.968,A -85,B 0,C 180,E1 -25002.177,E2 -25002.177} C_VEL
LIN {X 0,Y 148.715,Z 294.334,A -85,B 0,C 180,E1 -25003.528,E2 -25003.528} C_VEL
LIN {X 0,Y 145.832,Z 289.707,A -85,B 0,C 180,E1 -25010.814,E2 -25010.814} C_VEL
LIN {X 0,Y 145.491,Z 287.982,A -85,B 0,C 180,E1 -25013.064,E2 -25013.064} C_VEL
LIN {X 0,Y 144.52,Z 287.299,A -85,B 0,C 180,E1 -25020,E2 -25020} C_VEL
LIN {X 0,Y 145.499,Z 288.179,A -85,B 0,C 180,E1 -25027.808,E2 -25027.808} C_VEL
LIN {X 0,Y 146.068,Z 290.768,A -85,B 0,C 180,E1 -25031.097,E2 -25031.097} C_VEL
LIN {X 0,Y 148.404,Z 293.594,A -85,B 0,C 180,E1 -25036.508,E2 -25036.508} C_VEL
LIN {X 0,Y 149.618,Z 296.367,A -85,B 0,C 180,E1 -25039.197,E2 -25039.197} C_VEL
LIN {X 0,Y 151.213,Z 298.637,A -85,B 0,C 180,E1 -25041.828,E2 -25041.828} C_VEL
LIN {X 0,Y 153.715,Z 303.243,A -85,B 0,C 180,E1 -25045.744,E2 -25045.744} C_VEL
LIN {X 0,Y 155.847,Z 307.932,A -85,B 0,C 180,E1 -25048.998,E2 -25048.998} C_VEL
LIN {X 0,Y 158.191,Z 314.97,A -85,B 0,C 180,E1 -25052.973,E2 -25052.973} C_VEL
LIN {X 0,Y 159.893,Z 321.724,A -85,B 0,C 180,E1 -25056.353,E2 -25056.353} C_VEL
LIN {X 0,Y 160.676,Z 326.621,A -85,B 0,C 180,E1 -25058.556,E2 -25058.556} C_VEL
LIN {X 0,Y 160.771,Z 333.825,A -85,B 0,C 180,E1 -25061.451,E2 -25061.451} C_VEL
LIN {X 0,Y 159.738,Z 343.612,A -85,B 0,C 180,E1 -25065.255,E2 -25065.255} C_VEL
LIN {X 0,Y 159.093,Z 345.547,A -85,B 0,C 180,E1 -25065.912,E2 -25065.912} C_VEL
LIN {X 0,Y 153.07,Z 355.956,A -85,B 0,C 180,E1 -25069.136,E2 -25069.136} C_VEL
LIN {X 0,Y 147.542,Z 364.537,A -85,B 0,C 180,E1 -25072.603,E2 -25072.603} C_VEL
LIN {X 0,Y 141.697,Z 372.76,A -85,B 0,C 180,E1 -25076.935,E2 -25076.935} C_VEL
LIN {X 0,Y 137.552,Z 378.487,A -85,B 0,C 180,E1 -25080.962,E2 -25080.962} C_VEL
LIN {X 0,Y 134.025,Z 383.189,A -85,B 0,C 180,E1 -25085.197,E2 -25085.197} C_VEL
LIN {X 0,Y 130.286,Z 388.06,A -85,B 0,C 180,E1 -25091.116,E2 -25091.116} C_VEL
LIN {X 0,Y 127.888,Z 391.442,A -85,B 0,C 180,E1 -25097.302,E2 -25097.302} C_VEL
LIN {X 0,Y 126.666,Z 393.442,A -85,B 0,C 180,E1 -25103.629,E2 -25103.629} C_VEL
LIN {X 0,Y 126.391,Z 394.119,A -85,B 0,C 180,E1 -25110,E2 -25110} C_VEL
LIN {X 0,Y 126.666,Z 393.488,A -85,B 0,C 180,E1 -25116.372,E2 -25116.372} C_VEL
LIN {X 0,Y 127.881,Z 391.527,A -85,B 0,C 180,E1 -25122.699,E2 -25122.699} C_VEL
LIN {X 0,Y 130.23,Z 388.188,A -85,B 0,C 180,E1 -25128.893,E2 -25128.893} C_VEL
LIN {X 0,Y 133.979,Z 383.366,A -85,B 0,C 180,E1 -25134.813,E2 -25134.813} C_VEL
LIN {X 0,Y 138.726,Z 376.912,A -85,B 0,C 180,E1 -25140.439,E2 -25140.439} C_VEL
LIN {X 0,Y 144.001,Z 369.716,A -85,B 0,C 180,E1 -25144.993,E2 -25144.993} C_VEL
LIN {X 0,Y 149.244,Z 362.17,A -85,B 0,C 180,E1 -25148.606,E2 -25148.606} C_VEL
LIN {X 0,Y 154.877,Z 353.109,A -85,B 0,C 180,E1 -25152.015,E2 -25152.015} C_VEL
LIN {X 0,Y 158.999,Z 346.021,A -85,B 0,C 180,E1 -25154.121,E2 -25154.121} C_VEL
LIN {X 0,Y 159.806,Z 344.082,A -85,B 0,C 180,E1 -25154.722,E2 -25154.722} C_VEL
LIN {X 0,Y 160.883,Z 334.29,A -85,B 0,C 180,E1 -25158.542,E2 -25158.542} C_VEL
LIN {X 0,Y 160.787,Z 327.021,A -85,B 0,C 180,E1 -25161.476,E2 -25161.476} C_VEL
LIN {X 0,Y 159.761,Z 320.653,A -85,B 0,C 180,E1 -25164.376,E2 -25164.376} C_VEL
LIN {X 0,Y 157.601,Z 312.844,A -85,B 0,C 180,E1 -25168.4,E2 -25168.4} C_VEL
LIN {X 0,Y 155.296,Z 306.377,A -85,B 0,C 180,E1 -25172.239,E2 -25172.239} C_VEL
LIN {X 0,Y 153.128,Z 301.859,A -85,B 0,C 180,E1 -25175.602,E2 -25175.602} C_VEL
LIN {X 0,Y 150.718,Z 297.558,A -85,B 0,C 180,E1 -25179.529,E2 -25179.529} C_VEL
LIN {X 0,Y 149.167,Z 295.493,A -85,B 0,C 180,E1 -25182.166,E2 -25182.166} C_VEL
LIN {X 0,Y 148.615,Z 294.053,A -85,B 0,C 180,E1 -25183.516,E2 -25183.516} C_VEL
LIN {X 0,Y 146.307,Z 291.124,A -85,B 0,C 180,E1 -25188.922,E2 -25188.922} C_VEL
LIN {X 0,Y 145.596,Z 288.13,A -85,B 0,C 180,E1 -25193.069,E2 -25193.069} C_VEL
LIN {X 0,Y 144.811,Z 287.47,A -85,B 0,C 180,E1 -25200,E2 -25200} C_VEL
LIN {X 0,Y 145.689,Z 288.23,A -85,B 0,C 180,E1 -25206.752,E2 -25206.752} C_VEL
LIN {X 0,Y 146.551,Z 291.357,A -85,B 0,C 180,E1 -25211.059,E2 -25211.059} C_VEL
LIN {X 0,Y 147.673,Z 292.692,A -85,B 0,C 180,E1 -25213.766,E2 -25213.766} C_VEL
LIN {X 0,Y 148.91,Z 294.641,A -85,B 0,C 180,E1 -25216.45,E2 -25216.45} C_VEL
LIN {X 0,Y 150.157,Z 297.568,A -85,B 0,C 180,E1 -25219.125,E2 -25219.125} C_VEL
LIN {X 0,Y 151.008,Z 298.652,A -85,B 0,C 180,E1 -25220.429,E2 -25220.429} C_VEL
LIN {X 0,Y 152.332,Z 302.327,A -85,B 0,C 180,E1 -25223.087,E2 -25223.087} C_VEL
LIN {X 0,Y 153.246,Z 303.798,A -85,B 0,C 180,E1 -25224.377,E2 -25224.377} C_VEL
LIN {X 0,Y 156.357,Z 312.386,A -85,B 0,C 180,E1 -25229.632,E2 -25229.632} C_VEL
LIN {X 0,Y 158.556,Z 320.163,A -85,B 0,C 180,E1 -25233.646,E2 -25233.646} C_VEL
LIN {X 0,Y 159.842,Z 326.867,A -85,B 0,C 180,E1 -25236.695,E2 -25236.695} C_VEL
LIN {X 0,Y 160.104,Z 331.995,A -85,B 0,C 180,E1 -25238.721,E2 -25238.721} C_VEL
LIN {X 0,Y 159.512,Z 340.312,A -85,B 0,C 180,E1 -25241.751,E2 -25241.751} C_VEL
LIN {X 0,Y 158.076,Z 348.247,A -85,B 0,C 180,E1 -25244.654,E2 -25244.654} C_VEL
LIN {X 0,Y 157.012,Z 352.196,A -85,B 0,C 180,E1 -25246.107,E2 -25246.107} C_VEL
LIN {X 0,Y 151.061,Z 362.148,A -85,B 0,C 180,E1 -25249.357,E2 -25249.357} C_VEL
LIN {X 0,Y 145.583,Z 370.479,A -85,B 0,C 180,E1 -25252.883,E2 -25252.883} C_VEL
LIN {X 0,Y 139.938,Z 378.448,A -85,B 0,C 180,E1 -25257.324,E2 -25257.324} C_VEL
LIN {X 0,Y 135.3,Z 384.871,A -85,B 0,C 180,E1 -25262.128,E2 -25262.128} C_VEL
LIN {X 0,Y 131.186,Z 390.569,A -85,B 0,C 180,E1 -25267.975,E2 -25267.975} C_VEL
LIN {X 0,Y 128.219,Z 394.704,A -85,B 0,C 180,E1 -25274.094,E2 -25274.094} C_VEL
LIN {X 0,Y 126.68,Z 397.41,A -85,B 0,C 180,E1 -25280.419,E2 -25280.419} C_VEL
LIN {X 0,Y 126.39,Z 398.25,A -85,B 0,C 180,E1 -25283.614,E2 -25283.614} C_VEL
LIN {X 0,Y 126.361,Z 398.916,A -85,B 0,C 180,E1 -25290,E2 -25290} C_VEL
LIN {X 0,Y 126.371,Z 398.225,A -85,B 0,C 180,E1 -25296.386,E2 -25296.386} C_VEL
LIN {X 0,Y 127.311,Z 396.185,A -85,B 0,C 180,E1 -25302.757,E2 -25302.757} C_VEL
LIN {X 0,Y 129.491,Z 392.752,A -85,B 0,C 180,E1 -25309.004,E2 -25309.004} C_VEL
LIN {X 0,Y 133.091,Z 387.826,A -85,B 0,C 180,E1 -25314.989,E2 -25314.989} C_VEL
LIN {X 0,Y 136.513,Z 383.079,A -85,B 0,C 180,E1 -25319.278,E2 -25319.278} C_VEL
LIN {X 0,Y 141.471,Z 376.201,A -85,B 0,C 180,E1 -25323.978,E2 -25323.978} C_VEL
LIN {X 0,Y 147.28,Z 367.67,A -85,B 0,C 180,E1 -25328.341,E2 -25328.341} C_VEL
LIN {X 0,Y 153.028,Z 358.776,A -85,B 0,C 180,E1 -25331.754,E2 -25331.754} C_VEL
LIN {X 0,Y 156.964,Z 352.039,A -85,B 0,C 180,E1 -25333.863,E2 -25333.863} C_VEL
LIN {X 0,Y 158.784,Z 344.173,A -85,B 0,C 180,E1 -25336.755,E2 -25336.755} C_VEL
LIN {X 0,Y 159.767,Z 336.358,A -85,B 0,C 180,E1 -25339.601,E2 -25339.601} C_VEL
LIN {X 0,Y 159.983,Z 329.188,A -85,B 0,C 180,E1 -25342.254,E2 -25342.254} C_VEL
LIN {X 0,Y 159.108,Z 322.872,A -85,B 0,C 180,E1 -25344.955,E2 -25344.955} C_VEL
LIN {X 0,Y 157.057,Z 314.831,A -85,B 0,C 180,E1 -25348.88,E2 -25348.88} C_VEL
LIN {X 0,Y 154.602,Z 307.671,A -85,B 0,C 180,E1 -25352.962,E2 -25352.962} C_VEL
LIN {X 0,Y 153.262,Z 304.202,A -85,B 0,C 180,E1 -25355.214,E2 -25355.214} C_VEL
LIN {X 0,Y 151.867,Z 301.945,A -85,B 0,C 180,E1 -25357.181,E2 -25357.181} C_VEL
LIN {X 0,Y 150.086,Z 300.804,A -85,B 0,C 180,E1 -25359.284,E2 -25359.284} C_VEL
LIN {X 0,Y 145.479,Z 299.651,A -85,B 0,C 180,E1 -25365.277,E2 -25365.277} C_VEL
LIN {X 0,Y 144.732,Z 298.992,A -85,B 0,C 180,E1 -25366.828,E2 -25366.828} C_VEL
LIN {X 0,Y 143.009,Z 294.641,A -85,B 0,C 180,E1 -25374.36,E2 -25374.36} C_VEL
LIN {X 0,Y 142.409,Z 294.082,A -85,B 0,C 180,E1 -25380,E2 -25380} C_VEL
LIN {X 0,Y 142.846,Z 294.56,A -85,B 0,C 180,E1 -25385.647,E2 -25385.647} C_VEL
LIN {X 0,Y 143.238,Z 295.824,A -85,B 0,C 180,E1 -25388.465,E2 -25388.465} C_VEL
LIN {X 0,Y 145.823,Z 300.919,A -85,B 0,C 180,E1 -25396.809,E2 -25396.809} C_VEL
LIN {X 0,Y 147.687,Z 304.243,A -85,B 0,C 180,E1 -25400.709,E2 -25400.709} C_VEL
LIN {X 0,Y 149.979,Z 308.881,A -85,B 0,C 180,E1 -25404.945,E2 -25404.945} C_VEL
LIN {X 0,Y 151.848,Z 313.652,A -85,B 0,C 180,E1 -25408.433,E2 -25408.433} C_VEL
LIN {X 0,Y 153.606,Z 319.949,A -85,B 0,C 180,E1 -25412.192,E2 -25412.192} C_VEL
LIN {X 0,Y 155.047,Z 327.352,A -85,B 0,C 180,E1 -25416.105,E2 -25416.105} C_VEL
LIN {X 0,Y 155.379,Z 333.133,A -85,B 0,C 180,E1 -25418.765,E2 -25418.765} C_VEL
LIN {X 0,Y 154.786,Z 339.957,A -85,B 0,C 180,E1 -25421.602,E2 -25421.602} C_VEL
LIN {X 0,Y 153.89,Z 345.611,A -85,B 0,C 180,E1 -25423.966,E2 -25423.966} C_VEL
LIN {X 0,Y 152.823,Z 347.867,A -85,B 0,C 180,E1 -25424.68,E2 -25424.68} C_VEL
LIN {X 0,Y 146.761,Z 357.625,A -85,B 0,C 180,E1 -25427.9,E2 -25427.9} C_VEL
LIN {X 0,Y 141.007,Z 365.95,A -85,B 0,C 180,E1 -25431.463,E2 -25431.463} C_VEL
LIN {X 0,Y 134.981,Z 373.901,A -85,B 0,C 180,E1 -25435.965,E2 -25435.965} C_VEL
LIN {X 0,Y 130.038,Z 380.29,A -85,B 0,C 180,E1 -25440.895,E2 -25440.895} C_VEL
LIN {X 0,Y 126.451,Z 384.72,A -85,B 0,C 180,E1 -25445.365,E2 -25445.365} C_VEL
LIN {X 0,Y 123.548,Z 388.196,A -85,B 0,C 180,E1 -25450.044,E2 -25450.044} C_VEL
LIN {X 0,Y 120.971,Z 391.577,A -85,B 0,C 180,E1 -25456.563,E2 -25456.563} C_VEL
LIN {X 0,Y 119.602,Z 393.577,A -85,B 0,C 180,E1 -25463.251,E2 -25463.251} C_VEL
LIN {X 0,Y 119.365,Z 394.079,A -85,B 0,C 180,E1 -25466.625,E2 -25466.625} C_VEL
LIN {X 0,Y 119.294,Z 394.254,A -85,B 0,C 180,E1 -25470,E2 -25470} C_VEL
LIN {X 0,Y 119.365,Z 394.102,A -85,B 0,C 180,E1 -25473.376,E2 -25473.376} C_VEL
LIN {X 0,Y 120.12,Z 392.811,A -85,B 0,C 180,E1 -25480.11,E2 -25480.11} C_VEL
LIN {X 0,Y 122.097,Z 390.169,A -85,B 0,C 180,E1 -25486.727,E2 -25486.727} C_VEL
LIN {X 0,Y 125.309,Z 386.107,A -85,B 0,C 180,E1 -25493.117,E2 -25493.117} C_VEL
LIN {X 0,Y 128.756,Z 382.081,A -85,B 0,C 180,E1 -25497.644,E2 -25497.644} C_VEL
LIN {X 0,Y 132.605,Z 377.047,A -85,B 0,C 180,E1 -25502.006,E2 -25502.006} C_VEL
LIN {X 0,Y 138.224,Z 369.85,A -85,B 0,C 180,E1 -25506.686,E2 -25506.686} C_VEL
LIN {X 0,Y 143.754,Z 362.303,A -85,B 0,C 180,E1 -25510.375,E2 -25510.375} C_VEL
LIN {X 0,Y 149.674,Z 353.241,A -85,B 0,C 180,E1 -25513.836,E2 -25513.836} C_VEL
LIN {X 0,Y 153.991,Z 345.898,A -85,B 0,C 180,E1 -25516.082,E2 -25516.082} C_VEL
LIN {X 0,Y 155.216,Z 337.795,A -85,B 0,C 180,E1 -25519.467,E2 -25519.467} C_VEL
LIN {X 0,Y 155.475,Z 331.246,A -85,B 0,C 180,E1 -25522.278,E2 -25522.278} C_VEL
LIN {X 0,Y 154.951,Z 326.155,A -85,B 0,C 180,E1 -25524.728,E2 -25524.728} C_VEL
LIN {X 0,Y 153.443,Z 318.867,A -85,B 0,C 180,E1 -25528.629,E2 -25528.629} C_VEL
LIN {X 0,Y 151.299,Z 311.777,A -85,B 0,C 180,E1 -25533.07,E2 -25533.07} C_VEL
LIN {X 0,Y 149.443,Z 307.591,A -85,B 0,C 180,E1 -25536.438,E2 -25536.438} C_VEL
LIN {X 0,Y 147.351,Z 303.461,A -85,B 0,C 180,E1 -25540.496,E2 -25540.496} C_VEL
LIN {X 0,Y 144.952,Z 299.346,A -85,B 0,C 180,E1 -25545.97,E2 -25545.97} C_VEL
LIN {X 0,Y 143.158,Z 294.673,A -85,B 0,C 180,E1 -25554.365,E2 -25554.365} C_VEL
LIN {X 0,Y 142.693,Z 294.251,A -85,B 0,C 180,E1 -25560,E2 -25560} C_VEL
LIN {X 0,Y 143.307,Z 294.729,A -85,B 0,C 180,E1 -25565.629,E2 -25565.629} C_VEL
LIN {X 0,Y 146.013,Z 300.859,A -85,B 0,C 180,E1 -25575.707,E2 -25575.707} C_VEL
LIN {X 0,Y 147.639,Z 304.519,A -85,B 0,C 180,E1 -25579.464,E2 -25579.464} C_VEL
LIN {X 0,Y 149.557,Z 309.472,A -85,B 0,C 180,E1 -25583.543,E2 -25583.543} C_VEL
LIN {X 0,Y 151.921,Z 317.069,A -85,B 0,C 180,E1 -25588.482,E2 -25588.482} C_VEL
LIN {X 0,Y 153.592,Z 323.861,A -85,B 0,C 180,E1 -25592.274,E2 -25592.274} C_VEL
LIN {X 0,Y 154.596,Z 330.235,A -85,B 0,C 180,E1 -25595.424,E2 -25595.424} C_VEL
LIN {X 0,Y 154.684,Z 335.212,A -85,B 0,C 180,E1 -25597.545,E2 -25597.545} C_VEL
LIN {X 0,Y 153.722,Z 343.201,A -85,B 0,C 180,E1 -25600.676,E2 -25600.676} C_VEL
LIN {X 0,Y 151.796,Z 351.687,A -85,B 0,C 180,E1 -25603.986,E2 -25603.986} C_VEL
LIN {X 0,Y 151.275,Z 353.207,A -85,B 0,C 180,E1 -25604.589,E2 -25604.589} C_VEL
LIN {X 0,Y 144.727,Z 363.504,A -85,B 0,C 180,E1 -25608.109,E2 -25608.109} C_VEL
LIN {X 0,Y 139.061,Z 371.581,A -85,B 0,C 180,E1 -25611.749,E2 -25611.749} C_VEL
LIN {X 0,Y 133.207,Z 379.327,A -85,B 0,C 180,E1 -25616.359,E2 -25616.359} C_VEL
LIN {X 0,Y 129.017,Z 384.736,A -85,B 0,C 180,E1 -25620.642,E2 -25620.642} C_VEL
LIN {X 0,Y 124.583,Z 390.434,A -85,B 0,C 180,E1 -25626.741,E2 -25626.741} C_VEL
LIN {X 0,Y 121.356,Z 394.569,A -85,B 0,C 180,E1 -25633.168,E2 -25633.168} C_VEL
LIN {X 0,Y 119.66,Z 397.275,A -85,B 0,C 180,E1 -25639.851,E2 -25639.851} C_VEL
LIN {X 0,Y 119.149,Z 398.616,A -85,B 0,C 180,E1 -25646.618,E2 -25646.618} C_VEL
LIN {X 0,Y 119.277,Z 398.782,A -85,B 0,C 180,E1 -25650,E2 -25650} C_VEL
LIN {X 0,Y 119.286,Z 398.09,A -85,B 0,C 180,E1 -25656.767,E2 -25656.767} C_VEL
LIN {X 0,Y 120.36,Z 396.049,A -85,B 0,C 180,E1 -25663.507,E2 -25663.507} C_VEL
LIN {X 0,Y 122.78,Z 392.616,A -85,B 0,C 180,E1 -25670.086,E2 -25670.086} C_VEL
LIN {X 0,Y 126.652,Z 387.689,A -85,B 0,C 180,E1 -25676.354,E2 -25676.354} C_VEL
LIN {X 0,Y 131.716,Z 381.121,A -85,B 0,C 180,E1 -25682.247,E2 -25682.247} C_VEL
LIN {X 0,Y 137.267,Z 373.822,A -85,B 0,C 180,E1 -25686.984,E2 -25686.984} C_VEL
LIN {X 0,Y 143.704,Z 364.781,A -85,B 0,C 180,E1 -25691.317,E2 -25691.317} C_VEL
LIN {X 0,Y 149.859,Z 355.302,A -85,B 0,C 180,E1 -25694.705,E2 -25694.705} C_VEL
LIN {X 0,Y 151.207,Z 353.049,A -85,B 0,C 180,E1 -25695.386,E2 -25695.386} C_VEL
LIN {X 0,Y 152.992,Z 346.335,A -85,B 0,C 180,E1 -25698.039,E2 -25698.039} C_VEL
LIN {X 0,Y 154.253,Z 338.249,A -85,B 0,C 180,E1 -25701.164,E2 -25701.164} C_VEL
LIN {X 0,Y 154.591,Z 331.755,A -85,B 0,C 180,E1 -25703.772,E2 -25703.772} C_VEL
LIN {X 0,Y 153.825,Z 325.447,A -85,B 0,C 180,E1 -25706.753,E2 -25706.753} C_VEL
LIN {X 0,Y 151.981,Z 317.472,A -85,B 0,C 180,E1 -25711.103,E2 -25711.103} C_VEL
LIN {X 0,Y 150.696,Z 313.25,A -85,B 0,C 180,E1 -25713.701,E2 -25713.701} C_VEL
LIN {X 0,Y 149.375,Z 309.262,A -85,B 0,C 180,E1 -25716.427,E2 -25716.427} C_VEL
LIN {X 0,Y 147.436,Z 304.303,A -85,B 0,C 180,E1 -25720.508,E2 -25720.508} C_VEL
LIN {X 0,Y 145.457,Z 300.023,A -85,B 0,C 180,E1 -25725.09,E2 -25725.09} C_VEL
LIN {X 0,Y 144.732,Z 298.992,A -85,B 0,C 180,E1 -25726.828,E2 -25726.828} C_VEL
LIN {X 0,Y 143.7,Z 298.369,A -85,B 0,C 180,E1 -25729.133,E2 -25729.133} C_VEL
LIN {X 0,Y 141.766,Z 299.208,A -85,B 0,C 180,E1 -25733.035,E2 -25733.035} C_VEL
LIN {X 0,Y 140.129,Z 300.74,A -85,B 0,C 180,E1 -25737.865,E2 -25737.865} C_VEL
LIN {X 0,Y 139.988,Z 300.785,A -85,B 0,C 180,E1 -25739.507,E2 -25739.507} C_VEL
LIN {X 0,Y 140.354,Z 301.338,A -85,B 0,C 180,E1 -25745.748,E2 -25745.748} C_VEL
LIN {X 0,Y 141.983,Z 305.893,A -85,B 0,C 180,E1 -25754.33,E2 -25754.33} C_VEL
LIN {X 0,Y 144.154,Z 310.151,A -85,B 0,C 180,E1 -25759.955,E2 -25759.955} C_VEL
LIN {X 0,Y 146.255,Z 314.998,A -85,B 0,C 180,E1 -25764.615,E2 -25764.615} C_VEL
LIN {X 0,Y 147.563,Z 318.959,A -85,B 0,C 180,E1 -25767.669,E2 -25767.669} C_VEL
LIN {X 0,Y 149.065,Z 325.721,A -85,B 0,C 180,E1 -25771.935,E2 -25771.935} C_VEL
LIN {X 0,Y 149.947,Z 332.859,A -85,B 0,C 180,E1 -25775.879,E2 -25775.879} C_VEL
LIN {X 0,Y 149.727,Z 338.216,A -85,B 0,C 180,E1 -25778.404,E2 -25778.404} C_VEL
LIN {X 0,Y 148.596,Z 345.119,A -85,B 0,C 180,E1 -25781.464,E2 -25781.464} C_VEL
LIN {X 0,Y 148.243,Z 347.027,A -85,B 0,C 180,E1 -25782.32,E2 -25782.32} C_VEL
LIN {X 0,Y 147.548,Z 348.585,A -85,B 0,C 180,E1 -25782.896,E2 -25782.896} C_VEL
LIN {X 0,Y 141.563,Z 357.762,A -85,B 0,C 180,E1 -25785.97,E2 -25785.97} C_VEL
LIN {X 0,Y 135.533,Z 366.087,A -85,B 0,C 180,E1 -25789.595,E2 -25789.595} C_VEL
LIN {X 0,Y 129.14,Z 374.037,A -85,B 0,C 180,E1 -25794.195,E2 -25794.195} C_VEL
LIN {X 0,Y 123.845,Z 380.427,A -85,B 0,C 180,E1 -25799.287,E2 -25799.287} C_VEL
LIN {X 0,Y 120.03,Z 384.856,A -85,B 0,C 180,E1 -25803.951,E2 -25803.951} C_VEL
LIN {X 0,Y 116.861,Z 388.333,A -85,B 0,C 180,E1 -25808.849,E2 -25808.849} C_VEL
LIN {X 0,Y 114.052,Z 391.713,A -85,B 0,C 180,E1 -25815.731,E2 -25815.731} C_VEL
LIN {X 0,Y 112.564,Z 393.712,A -85,B 0,C 180,E1 -25822.827,E2 -25822.827} C_VEL
LIN {X 0,Y 112.208,Z 394.388,A -85,B 0,C 180,E1 -25830,E2 -25830} C_VEL
LIN {X 0,Y 112.564,Z 393.757,A -85,B 0,C 180,E1 -25837.174,E2 -25837.174} C_VEL
LIN {X 0,Y 114.043,Z 391.796,A -85,B 0,C 180,E1 -25844.271,E2 -25844.271} C_VEL
LIN {X 0,Y 116.807,Z 388.458,A -85,B 0,C 180,E1 -25851.162,E2 -25851.162} C_VEL
LIN {X 0,Y 121.208,Z 383.634,A -85,B 0,C 180,E1 -25857.637,E2 -25857.637} C_VEL
LIN {X 0,Y 126.329,Z 377.525,A -85,B 0,C 180,E1 -25863.437,E2 -25863.437} C_VEL
LIN {X 0,Y 132.591,Z 369.983,A -85,B 0,C 180,E1 -25868.522,E2 -25868.522} C_VEL
LIN {X 0,Y 139.406,Z 361.073,A -85,B 0,C 180,E1 -25872.89,E2 -25872.89} C_VEL
LIN {X 0,Y 145.735,Z 351.708,A -85,B 0,C 180,E1 -25876.334,E2 -25876.334} C_VEL
LIN {X 0,Y 148.343,Z 347.329,A -85,B 0,C 180,E1 -25877.715,E2 -25877.715} C_VEL
LIN {X 0,Y 149.653,Z 339.962,A -85,B 0,C 180,E1 -25880.993,E2 -25880.993} C_VEL
LIN {X 0,Y 150.081,Z 334.433,A -85,B 0,C 180,E1 -25883.539,E2 -25883.539} C_VEL
LIN {X 0,Y 149.618,Z 328.851,A -85,B 0,C 180,E1 -25886.501,E2 -25886.501} C_VEL
LIN {X 0,Y 148.401,Z 322.091,A -85,B 0,C 180,E1 -25890.533,E2 -25890.533} C_VEL
LIN {X 0,Y 146.905,Z 316.329,A -85,B 0,C 180,E1 -25894.496,E2 -25894.496} C_VEL
LIN {X 0,Y 144.908,Z 311.885,A -85,B 0,C 180,E1 -25898.669,E2 -25898.669} C_VEL
LIN {X 0,Y 143.201,Z 308.21,A -85,B 0,C 180,E1 -25902.874,E2 -25902.874} C_VEL
LIN {X 0,Y 142.23,Z 306.145,A -85,B 0,C 180,E1 -25905.696,E2 -25905.696} C_VEL
LIN {X 0,Y 140.646,Z 301.487,A -85,B 0,C 180,E1 -25914.264,E2 -25914.264} C_VEL
LIN {X 0,Y 140.259,Z 300.924,A -85,B 0,C 180,E1 -25920,E2 -25920} C_VEL
LIN {X 0,Y 140.794,Z 301.61,A -85,B 0,C 180,E1 -25925.729,E2 -25925.729} C_VEL
LIN {X 0,Y 142.622,Z 306.5,A -85,B 0,C 180,E1 -25934.263,E2 -25934.263} C_VEL
LIN {X 0,Y 144.082,Z 310.256,A -85,B 0,C 180,E1 -25938.485,E2 -25938.485} C_VEL
LIN {X 0,Y 145.679,Z 315.048,A -85,B 0,C 180,E1 -25942.702,E2 -25942.702} C_VEL
LIN {X 0,Y 147.536,Z 322.214,A -85,B 0,C 180,E1 -25947.674,E2 -25947.674} C_VEL
LIN {X 0,Y 148.829,Z 329.239,A -85,B 0,C 180,E1 -25951.788,E2 -25951.788} C_VEL
LIN {X 0,Y 149.401,Z 335.883,A -85,B 0,C 180,E1 -25955.227,E2 -25955.227} C_VEL
LIN {X 0,Y 148.48,Z 343.357,A -85,B 0,C 180,E1 -25958.417,E2 -25958.417} C_VEL
LIN {X 0,Y 146.613,Z 351.219,A -85,B 0,C 180,E1 -25961.663,E2 -25961.663} C_VEL
LIN {X 0,Y 145.638,Z 354.209,A -85,B 0,C 180,E1 -25962.94,E2 -25962.94} C_VEL
LIN {X 0,Y 139.498,Z 363.371,A -85,B 0,C 180,E1 -25966.153,E2 -25966.153} C_VEL
LIN {X 0,Y 133.526,Z 371.447,A -85,B 0,C 180,E1 -25969.851,E2 -25969.851} C_VEL
LIN {X 0,Y 127.31,Z 379.192,A -85,B 0,C 180,E1 -25974.574,E2 -25974.574} C_VEL
LIN {X 0,Y 122.451,Z 385.042,A -85,B 0,C 180,E1 -25979.419,E2 -25979.419} C_VEL
LIN {X 0,Y 118.032,Z 390.299,A -85,B 0,C 180,E1 -25985.367,E2 -25985.367} C_VEL
LIN {X 0,Y 114.532,Z 394.434,A -85,B 0,C 180,E1 -25992.132,E2 -25992.132} C_VEL
LIN {X 0,Y 112.663,Z 397.141,A -85,B 0,C 180,E1 -25999.214,E2 -25999.214} C_VEL
LIN {X 0,Y 112.056,Z 398.481,A -85,B 0,C 180,E1 -26006.404,E2 -26006.404} C_VEL
LIN {X 0,Y 112.195,Z 398.647,A -85,B 0,C 180,E1 -26010,E2 -26010} C_VEL
LIN {X 0,Y 112.225,Z 397.954,A -85,B 0,C 180,E1 -26017.195,E2 -26017.195} C_VEL
LIN {X 0,Y 113.416,Z 395.913,A -85,B 0,C 180,E1 -26024.351,E2 -26024.351} C_VEL
LIN {X 0,Y 116.116,Z 392.48,A -85,B 0,C 180,E1 -26031.294,E2 -26031.294} C_VEL
LIN {X 0,Y 120.293,Z 387.552,A -85,B 0,C 180,E1 -26037.865,E2 -26037.865} C_VEL
LIN {X 0,Y 125.732,Z 380.984,A -85,B 0,C 180,E1 -26043.984,E2 -26043.984} C_VEL
LIN {X 0,Y 131.631,Z 373.685,A -85,B 0,C 180,E1 -26048.855,E2 -26048.855} C_VEL
LIN {X 0,Y 138.441,Z 364.644,A -85,B 0,C 180,E1 -26053.261,E2 -26053.261} C_VEL
LIN {X 0,Y 144.877,Z 355.164,A -85,B 0,C 180,E1 -26056.69,E2 -26056.69} C_VEL
LIN {X 0,Y 145.558,Z 354.059,A -85,B 0,C 180,E1 -26057.031,E2 -26057.031} C_VEL
LIN {X 0,Y 147.652,Z 346.534,A -85,B 0,C 180,E1 -26060.208,E2 -26060.208} C_VEL
LIN {X 0,Y 149.042,Z 339.007,A -85,B 0,C 180,E1 -26063.286,E2 -26063.286} C_VEL
LIN {X 0,Y 149.233,Z 333.946,A -85,B 0,C 180,E1 -26065.589,E2 -26065.589} C_VEL
LIN {X 0,Y 148.599,Z 328.13,A -85,B 0,C 180,E1 -26068.652,E2 -26068.652} C_VEL
LIN {X 0,Y 147.392,Z 322.003,A -85,B 0,C 180,E1 -26072.296,E2 -26072.296} C_VEL
LIN {X 0,Y 145.834,Z 316.24,A -85,B 0,C 180,E1 -26076.297,E2 -26076.297} C_VEL
LIN {X 0,Y 145.509,Z 314.833,A -85,B 0,C 180,E1 -26077.27,E2 -26077.27} C_VEL
LIN {X 0,Y 143.883,Z 310.047,A -85,B 0,C 180,E1 -26081.489,E2 -26081.489} C_VEL
LIN {X 0,Y 142.426,Z 306.252,A -85,B 0,C 180,E1 -26085.716,E2 -26085.716} C_VEL
LIN {X 0,Y 140.529,Z 301.449,A -85,B 0,C 180,E1 -26094.26,E2 -26094.26} C_VEL
LIN {X 0,Y 139.988,Z 300.785,A -85,B 0,C 180,E1 -26099.507,E2 -26099.507} C_VEL
LIN {X 0,Y 139.884,Z 301.034,A -85,B 0,C 180,E1 -26101.109,E2 -26101.109} C_VEL
LIN {X 0,Y 139.464,Z 302.581,A -85,B 0,C 180,E1 -26103.448,E2 -26103.448} C_VEL
LIN {X 0,Y 138.038,Z 310.001,A -85,B 0,C 180,E1 -26110.295,E2 -26110.295} C_VEL
LIN {X 0,Y 138.192,Z 311.127,A -85,B 0,C 180,E1 -26111.91,E2 -26111.91} C_VEL
LIN {X 0,Y 138.947,Z 312.58,A -85,B 0,C 180,E1 -26114.65,E2 -26114.65} C_VEL
LIN {X 0,Y 140.82,Z 317.073,A -85,B 0,C 180,E1 -26120.448,E2 -26120.448} C_VEL
LIN {X 0,Y 142.293,Z 320.963,A -85,B 0,C 180,E1 -26124.311,E2 -26124.311} C_VEL
LIN {X 0,Y 143.231,Z 324.562,A -85,B 0,C 180,E1 -26127.211,E2 -26127.211} C_VEL
LIN {X 0,Y 144.257,Z 331.155,A -85,B 0,C 180,E1 -26131.583,E2 -26131.583} C_VEL
LIN {X 0,Y 144.618,Z 336.666,A -85,B 0,C 180,E1 -26134.821,E2 -26134.821} C_VEL
LIN {X 0,Y 144.105,Z 341.775,A -85,B 0,C 180,E1 -26137.389,E2 -26137.389} C_VEL
LIN {X 0,Y 142.658,Z 348.408,A -85,B 0,C 180,E1 -26140.54,E2 -26140.54} C_VEL
LIN {X 0,Y 142.364,Z 349.307,A -85,B 0,C 180,E1 -26140.956,E2 -26140.956} C_VEL
LIN {X 0,Y 135.449,Z 359.38,A -85,B 0,C 180,E1 -26144.485,E2 -26144.485} C_VEL
LIN {X 0,Y 129.159,Z 367.451,A -85,B 0,C 180,E1 -26148.198,E2 -26148.198} C_VEL
LIN {X 0,Y 122.544,Z 375.177,A -85,B 0,C 180,E1 -26152.974,E2 -26152.974} C_VEL
LIN {X 0,Y 117.764,Z 380.564,A -85,B 0,C 180,E1 -26157.513,E2 -26157.513} C_VEL
LIN {X 0,Y 113.678,Z 384.992,A -85,B 0,C 180,E1 -26162.376,E2 -26162.376} C_VEL
LIN {X 0,Y 110.235,Z 388.469,A -85,B 0,C 180,E1 -26167.51,E2 -26167.51} C_VEL
LIN {X 0,Y 107.169,Z 391.848,A -85,B 0,C 180,E1 -26174.793,E2 -26174.793} C_VEL
LIN {X 0,Y 105.516,Z 393.847,A -85,B 0,C 180,E1 -26182.345,E2 -26182.345} C_VEL
LIN {X 0,Y 105.199,Z 394.349,A -85,B 0,C 180,E1 -26186.17,E2 -26186.17} C_VEL
LIN {X 0,Y 105.114,Z 394.523,A -85,B 0,C 180,E1 -26190,E2 -26190} C_VEL
LIN {X 0,Y 105.199,Z 394.371,A -85,B 0,C 180,E1 -26193.831,E2 -26193.831} C_VEL
LIN {X 0,Y 106.151,Z 393.08,A -85,B 0,C 180,E1 -26201.457,E2 -26201.457} C_VEL
LIN {X 0,Y 108.501,Z 390.438,A -85,B 0,C 180,E1 -26208.898,E2 -26208.898} C_VEL
LIN {X 0,Y 112.38,Z 386.374,A -85,B 0,C 180,E1 -26215.962,E2 -26215.962} C_VEL
LIN {X 0,Y 116.292,Z 382.349,A -85,B 0,C 180,E1 -26220.911,E2 -26220.911} C_VEL
LIN {X 0,Y 120.752,Z 377.314,A -85,B 0,C 180,E1 -26225.593,E2 -26225.593} C_VEL
LIN {X 0,Y 127.093,Z 370.116,A -85,B 0,C 180,E1 -26230.524,E2 -26230.524} C_VEL
LIN {X 0,Y 134.287,Z 361.205,A -85,B 0,C 180,E1 -26234.954,E2 -26234.954} C_VEL
LIN {X 0,Y 140.934,Z 351.84,A -85,B 0,C 180,E1 -26238.419,E2 -26238.419} C_VEL
LIN {X 0,Y 142.37,Z 349.653,A -85,B 0,C 180,E1 -26239.083,E2 -26239.083} C_VEL
LIN {X 0,Y 143.974,Z 343.41,A -85,B 0,C 180,E1 -26242.011,E2 -26242.011} C_VEL
LIN {X 0,Y 144.638,Z 338.665,A -85,B 0,C 180,E1 -26244.332,E2 -26244.332} C_VEL
LIN {X 0,Y 144.61,Z 334.269,A -85,B 0,C 180,E1 -26246.771,E2 -26246.771} C_VEL
LIN {X 0,Y 143.913,Z 327.872,A -85,B 0,C 180,E1 -26250.767,E2 -26250.767} C_VEL
LIN {X 0,Y 142.667,Z 321.627,A -85,B 0,C 180,E1 -26255.326,E2 -26255.326} C_VEL
LIN {X 0,Y 141,Z 317.398,A -85,B 0,C 180,E1 -26259.579,E2 -26259.579} C_VEL
LIN {X 0,Y 139.569,Z 313.892,A -85,B 0,C 180,E1 -26263.921,E2 -26263.921} C_VEL
LIN {X 0,Y 138.376,Z 311.309,A -85,B 0,C 180,E1 -26268.278,E2 -26268.278} C_VEL
LIN {X 0,Y 137.804,Z 308.19,A -85,B 0,C 180,E1 -26274.145,E2 -26274.145} C_VEL
LIN {X 0,Y 137.578,Z 307.609,A -85,B 0,C 180,E1 -26277.072,E2 -26277.072} C_VEL
LIN {X 0,Y 137.52,Z 307.46,A -85,B 0,C 180,E1 -26280,E2 -26280} C_VEL
LIN {X 0,Y 137.652,Z 307.693,A -85,B 0,C 180,E1 -26282.926,E2 -26282.926} C_VEL
LIN {X 0,Y 137.948,Z 308.369,A -85,B 0,C 180,E1 -26285.848,E2 -26285.848} C_VEL
LIN {X 0,Y 139.533,Z 313.373,A -85,B 0,C 180,E1 -26294.586,E2 -26294.586} C_VEL
LIN {X 0,Y 140.694,Z 317.229,A -85,B 0,C 180,E1 -26298.795,E2 -26298.795} C_VEL
LIN {X 0,Y 141.629,Z 320.491,A -85,B 0,C 180,E1 -26301.849,E2 -26301.849} C_VEL
LIN {X 0,Y 142.818,Z 326.466,A -85,B 0,C 180,E1 -26306.288,E2 -26306.288} C_VEL
LIN {X 0,Y 143.695,Z 332.33,A -85,B 0,C 180,E1 -26310.087,E2 -26310.087} C_VEL
LIN {X 0,Y 144.055,Z 337.919,A -85,B 0,C 180,E1 -26313.288,E2 -26313.288} C_VEL
LIN {X 0,Y 143.586,Z 342.49,A -85,B 0,C 180,E1 -26315.489,E2 -26315.489} C_VEL
LIN {X 0,Y 141.895,Z 349.775,A -85,B 0,C 180,E1 -26318.725,E2 -26318.725} C_VEL
LIN {X 0,Y 140.062,Z 355.291,A -85,B 0,C 180,E1 -26321.177,E2 -26321.177} C_VEL
LIN {X 0,Y 133.36,Z 364.726,A -85,B 0,C 180,E1 -26324.647,E2 -26324.647} C_VEL
LIN {X 0,Y 127.162,Z 372.549,A -85,B 0,C 180,E1 -26328.454,E2 -26328.454} C_VEL
LIN {X 0,Y 121.562,Z 379.058,A -85,B 0,C 180,E1 -26332.623,E2 -26332.623} C_VEL
LIN {X 0,Y 115.954,Z 385.343,A -85,B 0,C 180,E1 -26338.053,E2 -26338.053} C_VEL
LIN {X 0,Y 111.562,Z 390.164,A -85,B 0,C 180,E1 -26343.833,E2 -26343.833} C_VEL
LIN {X 0,Y 107.753,Z 394.299,A -85,B 0,C 180,E1 -26350.966,E2 -26350.966} C_VEL
LIN {X 0,Y 105.658,Z 397.006,A -85,B 0,C 180,E1 -26358.489,E2 -26358.489} C_VEL
LIN {X 0,Y 104.96,Z 398.346,A -85,B 0,C 180,E1 -26366.16,E2 -26366.16} C_VEL
LIN {X 0,Y 105.102,Z 398.513,A -85,B 0,C 180,E1 -26370,E2 -26370} C_VEL
LIN {X 0,Y 105.164,Z 397.819,A -85,B 0,C 180,E1 -26377.681,E2 -26377.681} C_VEL
LIN {X 0,Y 106.51,Z 395.777,A -85,B 0,C 180,E1 -26385.304,E2 -26385.304} C_VEL
LIN {X 0,Y 109.483,Z 392.343,A -85,B 0,C 180,E1 -26392.653,E2 -26392.653} C_VEL
LIN {X 0,Y 114.017,Z 387.415,A -85,B 0,C 180,E1 -26399.545,E2 -26399.545} C_VEL
LIN {X 0,Y 119.87,Z 380.847,A -85,B 0,C 180,E1 -26405.895,E2 -26405.895} C_VEL
LIN {X 0,Y 126.153,Z 373.548,A -85,B 0,C 180,E1 -26410.889,E2 -26410.889} C_VEL
LIN {X 0,Y 132.25,Z 365.9,A -85,B 0,C 180,E1 -26414.759,E2 -26414.759} C_VEL
LIN {X 0,Y 138.928,Z 356.73,A -85,B 0,C 180,E1 -26418.259,E2 -26418.259} C_VEL
LIN {X 0,Y 140.019,Z 355.024,A -85,B 0,C 180,E1 -26418.842,E2 -26418.842} C_VEL
LIN {X 0,Y 142.325,Z 347.508,A -85,B 0,C 180,E1 -26422.193,E2 -26422.193} C_VEL
LIN {X 0,Y 143.702,Z 341.036,A -85,B 0,C 180,E1 -26425.072,E2 -26425.072} C_VEL
LIN {X 0,Y 143.902,Z 336.244,A -85,B 0,C 180,E1 -26427.505,E2 -26427.505} C_VEL
LIN {X 0,Y 143.283,Z 329.501,A -85,B 0,C 180,E1 -26431.509,E2 -26431.509} C_VEL
LIN {X 0,Y 142.171,Z 323.521,A -85,B 0,C 180,E1 -26435.648,E2 -26435.648} C_VEL
LIN {X 0,Y 141.471,Z 320.271,A -85,B 0,C 180,E1 -26438.125,E2 -26438.125} C_VEL
LIN {X 0,Y 140.149,Z 315.668,A -85,B 0,C 180,E1 -26442.49,E2 -26442.49} C_VEL
LIN {X 0,Y 139.342,Z 313.148,A -85,B 0,C 180,E1 -26445.393,E2 -26445.393} C_VEL
LIN {X 0,Y 137.712,Z 308.166,A -85,B 0,C 180,E1 -26454.142,E2 -26454.142} C_VEL
LIN {X 0,Y 137.26,Z 307.283,A -85,B 0,C 180,E1 -26460,E2 -26460} C_VEL
LIN {X 0,Y 137.544,Z 307.991,A -85,B 0,C 180,E1 -26465.866,E2 -26465.866} C_VEL
LIN {X 0,Y 138.192,Z 311.127,A -85,B 0,C 180,E1 -26471.91,E2 -26471.91} C_VEL
LIN {X 0,Y 138.487,Z 312.999,A -85,B 0,C 180,E1 -26474.227,E2 -26474.227} C_VEL
LIN {X 0,Y 138.425,Z 315.751,A -85,B 0,C 180,E1 -26476.404,E2 -26476.404} C_VEL
LIN {X 0,Y 137.75,Z 324.377,A -85,B 0,C 180,E1 -26482.047,E2 -26482.047} C_VEL
LIN {X 0,Y 137.952,Z 326.229,A -85,B 0,C 180,E1 -26483.534,E2 -26483.534} C_VEL
LIN {X 0,Y 138.735,Z 330.533,A -85,B 0,C 180,E1 -26487.124,E2 -26487.124} C_VEL
LIN {X 0,Y 139.196,Z 335.877,A -85,B 0,C 180,E1 -26490.871,E2 -26490.871} C_VEL
LIN {X 0,Y 139.108,Z 341.713,A -85,B 0,C 180,E1 -26494.467,E2 -26494.467} C_VEL
LIN {X 0,Y 137.747,Z 348.066,A -85,B 0,C 180,E1 -26497.753,E2 -26497.753} C_VEL
LIN {X 0,Y 137.205,Z 349.823,A -85,B 0,C 180,E1 -26498.652,E2 -26498.652} C_VEL
LIN {X 0,Y 136.392,Z 351.562,A -85,B 0,C 180,E1 -26499.384,E2 -26499.384} C_VEL
LIN {X 0,Y 129.421,Z 360.997,A -85,B 0,C 180,E1 -26502.854,E2 -26502.854} C_VEL
LIN {X 0,Y 121.833,Z 369.992,A -85,B 0,C 180,E1 -26507.328,E2 -26507.328} C_VEL
LIN {X 0,Y 115.11,Z 377.237,A -85,B 0,C 180,E1 -26512.371,E2 -26512.371} C_VEL
LIN {X 0,Y 108.852,Z 383.734,A -85,B 0,C 180,E1 -26518.901,E2 -26518.901} C_VEL
LIN {X 0,Y 103.682,Z 388.605,A -85,B 0,C 180,E1 -26526.002,E2 -26526.002} C_VEL
LIN {X 0,Y 100.326,Z 391.984,A -85,B 0,C 180,E1 -26533.728,E2 -26533.728} C_VEL
LIN {X 0,Y 98.495,Z 393.982,A -85,B 0,C 180,E1 -26541.796,E2 -26541.796} C_VEL
LIN {X 0,Y 98.014,Z 394.658,A -85,B 0,C 180,E1 -26550,E2 -26550} C_VEL
LIN {X 0,Y 98.495,Z 394.025,A -85,B 0,C 180,E1 -26558.205,E2 -26558.205} C_VEL
LIN {X 0,Y 100.316,Z 392.065,A -85,B 0,C 180,E1 -26566.275,E2 -26566.275} C_VEL
LIN {X 0,Y 103.633,Z 388.727,A -85,B 0,C 180,E1 -26574.011,E2 -26574.011} C_VEL
LIN {X 0,Y 108.78,Z 383.902,A -85,B 0,C 180,E1 -26581.122,E2 -26581.122} C_VEL
LIN {X 0,Y 115.034,Z 377.448,A -85,B 0,C 180,E1 -26587.659,E2 -26587.659} C_VEL
LIN {X 0,Y 121.773,Z 370.25,A -85,B 0,C 180,E1 -26592.699,E2 -26592.699} C_VEL
LIN {X 0,Y 129.356,Z 361.338,A -85,B 0,C 180,E1 -26597.178,E2 -26597.178} C_VEL
LIN {X 0,Y 136.321,Z 351.972,A -85,B 0,C 180,E1 -26600.654,E2 -26600.654} C_VEL
LIN {X 0,Y 137.297,Z 350.114,A -85,B 0,C 180,E1 -26601.378,E2 -26601.378} C_VEL
LIN {X 0,Y 138.941,Z 343.62,A -85,B 0,C 180,E1 -26604.719,E2 -26604.719} C_VEL
LIN {X 0,Y 139.347,Z 339.335,A -85,B 0,C 180,E1 -26607.168,E2 -26607.168} C_VEL
LIN {X 0,Y 139.084,Z 332.513,A -85,B 0,C 180,E1 -26611.701,E2 -26611.701} C_VEL
LIN {X 0,Y 138.26,Z 326.774,A -85,B 0,C 180,E1 -26616.202,E2 -26616.202} C_VEL
LIN {X 0,Y 136.929,Z 322.787,A -85,B 0,C 180,E1 -26620.511,E2 -26620.511} C_VEL
LIN {X 0,Y 135.765,Z 319.455,A -85,B 0,C 180,E1 -26624.999,E2 -26624.999} C_VEL
LIN {X 0,Y 134.633,Z 314.764,A -85,B 0,C 180,E1 -26634.007,E2 -26634.007} C_VEL
LIN {X 0,Y 134.515,Z 314.02,A -85,B 0,C 180,E1 -26637.005,E2 -26637.005} C_VEL
LIN {X 0,Y 134.472,Z 313.866,A -85,B 0,C 180,E1 -26640,E2 -26640} C_VEL
LIN {X 0,Y 134.59,Z 314.126,A -85,B 0,C 180,E1 -26642.993,E2 -26642.993} C_VEL
LIN {X 0,Y 134.787,Z 314.965,A -85,B 0,C 180,E1 -26645.986,E2 -26645.986} C_VEL
LIN {X 0,Y 135.792,Z 319.02,A -85,B 0,C 180,E1 -26653.468,E2 -26653.468} C_VEL
LIN {X 0,Y 136.742,Z 322.767,A -85,B 0,C 180,E1 -26657.961,E2 -26657.961} C_VEL
LIN {X 0,Y 137.415,Z 325.787,A -85,B 0,C 180,E1 -26660.978,E2 -26660.978} C_VEL
LIN {X 0,Y 138.217,Z 331.651,A -85,B 0,C 180,E1 -26665.607,E2 -26665.607} C_VEL
LIN {X 0,Y 138.668,Z 336.59,A -85,B 0,C 180,E1 -26669.026,E2 -26669.026} C_VEL
LIN {X 0,Y 138.732,Z 341.621,A -85,B 0,C 180,E1 -26672.133,E2 -26672.133} C_VEL
LIN {X 0,Y 137.861,Z 346.496,A -85,B 0,C 180,E1 -26674.6,E2 -26674.6} C_VEL
LIN {X 0,Y 135.767,Z 353.349,A -85,B 0,C 180,E1 -26677.87,E2 -26677.87} C_VEL
LIN {X 0,Y 134.621,Z 356.28,A -85,B 0,C 180,E1 -26679.24,E2 -26679.24} C_VEL
LIN {X 0,Y 128.454,Z 364.593,A -85,B 0,C 180,E1 -26682.386,E2 -26682.386} C_VEL
LIN {X 0,Y 121.891,Z 372.415,A -85,B 0,C 180,E1 -26686.219,E2 -26686.219} C_VEL
LIN {X 0,Y 115.959,Z 378.924,A -85,B 0,C 180,E1 -26690.477,E2 -26690.477} C_VEL
LIN {X 0,Y 109.634,Z 385.557,A -85,B 0,C 180,E1 -26696.444,E2 -26696.444} C_VEL
LIN {X 0,Y 105.186,Z 390.029,A -85,B 0,C 180,E1 -26702.114,E2 -26702.114} C_VEL
LIN {X 0,Y 101.024,Z 394.164,A -85,B 0,C 180,E1 -26709.644,E2 -26709.644} C_VEL
LIN {X 0,Y 98.683,Z 396.871,A -85,B 0,C 180,E1 -26717.663,E2 -26717.663} C_VEL
LIN {X 0,Y 97.886,Z 398.212,A -85,B 0,C 180,E1 -26725.882,E2 -26725.882} C_VEL
LIN {X 0,Y 98,Z 398.378,A -85,B 0,C 180,E1 -26730,E2 -26730} C_VEL
LIN {X 0,Y 98.107,Z 397.684,A -85,B 0,C 180,E1 -26738.237,E2 -26738.237} C_VEL
LIN {X 0,Y 99.646,Z 395.641,A -85,B 0,C 180,E1 -26746.386,E2 -26746.386} C_VEL
LIN {X 0,Y 102.926,Z 392.207,A -85,B 0,C 180,E1 -26754.185,E2 -26754.185} C_VEL
LIN {X 0,Y 107.828,Z 387.278,A -85,B 0,C 180,E1 -26761.427,E2 -26761.427} C_VEL
LIN {X 0,Y 114.156,Z 380.71,A -85,B 0,C 180,E1 -26767.999,E2 -26767.999} C_VEL
LIN {X 0,Y 120.851,Z 373.411,A -85,B 0,C 180,E1 -26773.103,E2 -26773.103} C_VEL
LIN {X 0,Y 127.298,Z 365.763,A -85,B 0,C 180,E1 -26777.014,E2 -26777.014} C_VEL
LIN {X 0,Y 133.821,Z 357.222,A -85,B 0,C 180,E1 -26780.315,E2 -26780.315} C_VEL
LIN {X 0,Y 134.527,Z 356.186,A -85,B 0,C 180,E1 -26780.697,E2 -26780.697} C_VEL
LIN {X 0,Y 136.894,Z 349.331,A -85,B 0,C 180,E1 -26783.957,E2 -26783.957} C_VEL
LIN {X 0,Y 138.068,Z 345.103,A -85,B 0,C 180,E1 -26785.95,E2 -26785.95} C_VEL
LIN {X 0,Y 138.608,Z 341.459,A -85,B 0,C 180,E1 -26787.835,E2 -26787.835} C_VEL
LIN {X 0,Y 138.547,Z 336.171,A -85,B 0,C 180,E1 -26791.086,E2 -26791.086} C_VEL
LIN {X 0,Y 137.967,Z 330.384,A -85,B 0,C 180,E1 -26795.15,E2 -26795.15} C_VEL
LIN {X 0,Y 137.26,Z 325.577,A -85,B 0,C 180,E1 -26798.997,E2 -26798.997} C_VEL
LIN {X 0,Y 136.248,Z 321.136,A -85,B 0,C 180,E1 -26803.519,E2 -26803.519} C_VEL
LIN {X 0,Y 135.611,Z 318.798,A -85,B 0,C 180,E1 -26806.514,E2 -26806.514} C_VEL
LIN {X 0,Y 134.576,Z 314.739,A -85,B 0,C 180,E1 -26814.005,E2 -26814.005} C_VEL
LIN {X 0,Y 134.326,Z 313.994,A -85,B 0,C 180,E1 -26817.001,E2 -26817.001} C_VEL
LIN {X 0,Y 134.22,Z 313.697,A -85,B 0,C 180,E1 -26820,E2 -26820} C_VEL
LIN {X 0,Y 134.398,Z 314.543,A -85,B 0,C 180,E1 -26826.003,E2 -26826.003} C_VEL
LIN {X 0,Y 135.555,Z 319.196,A -85,B 0,C 180,E1 -26835.025,E2 -26835.025} C_VEL
LIN {X 0,Y 136.752,Z 322.491,A -85,B 0,C 180,E1 -26839.515,E2 -26839.515} C_VEL
LIN {X 0,Y 137.952,Z 326.229,A -85,B 0,C 180,E1 -26843.534,E2 -26843.534} C_VEL
LIN {X 0,Y 138.07,Z 329.21,A -85,B 0,C 180,E1 -26845.655,E2 -26845.655} C_VEL
LIN {X 0,Y 137.159,Z 334.164,A -85,B 0,C 180,E1 -26848.21,E2 -26848.21} C_VEL
LIN {X 0,Y 134.976,Z 341.022,A -85,B 0,C 180,E1 -26851.249,E2 -26851.249} C_VEL
LIN {X 0,Y 133.409,Z 346.197,A -85,B 0,C 180,E1 -26853.843,E2 -26853.843} C_VEL
LIN {X 0,Y 131.742,Z 351.708,A -85,B 0,C 180,E1 -26856.851,E2 -26856.851} C_VEL
LIN {X 0,Y 129.516,Z 355.022,A -85,B 0,C 180,E1 -26858.111,E2 -26858.111} C_VEL
LIN {X 0,Y 122.348,Z 363.875,A -85,B 0,C 180,E1 -26861.69,E2 -26861.69} C_VEL
LIN {X 0,Y 114.57,Z 372.351,A -85,B 0,C 180,E1 -26866.362,E2 -26866.362} C_VEL
LIN {X 0,Y 107.545,Z 379.373,A -85,B 0,C 180,E1 -26871.892,E2 -26871.892} C_VEL
LIN {X 0,Y 101.269,Z 385.265,A -85,B 0,C 180,E1 -26878.635,E2 -26878.635} C_VEL
LIN {X 0,Y 97.21,Z 388.741,A -85,B 0,C 180,E1 -26884.292,E2 -26884.292} C_VEL
LIN {X 0,Y 93.501,Z 392.12,A -85,B 0,C 180,E1 -26892.503,E2 -26892.503} C_VEL
LIN {X 0,Y 91.454,Z 394.118,A -85,B 0,C 180,E1 -26901.159,E2 -26901.159} C_VEL
LIN {X 0,Y 90.941,Z 394.792,A -85,B 0,C 180,E1 -26910,E2 -26910} C_VEL
LIN {X 0,Y 91.454,Z 394.16,A -85,B 0,C 180,E1 -26918.842,E2 -26918.842} C_VEL
LIN {X 0,Y 93.489,Z 392.199,A -85,B 0,C 180,E1 -26927.5,E2 -26927.5} C_VEL
LIN {X 0,Y 97.164,Z 388.861,A -85,B 0,C 180,E1 -26935.722,E2 -26935.722} C_VEL
LIN {X 0,Y 102.735,Z 384.037,A -85,B 0,C 180,E1 -26943.181,E2 -26943.181} C_VEL
LIN {X 0,Y 109.48,Z 377.582,A -85,B 0,C 180,E1 -26949.937,E2 -26949.937} C_VEL
LIN {X 0,Y 116.655,Z 370.383,A -85,B 0,C 180,E1 -26955.064,E2 -26955.064} C_VEL
LIN {X 0,Y 124.635,Z 361.47,A -85,B 0,C 180,E1 -26959.575,E2 -26959.575} C_VEL
LIN {X 0,Y 131.788,Z 352.108,A -85,B 0,C 180,E1 -26963.124,E2 -26963.124} C_VEL
LIN {X 0,Y 133.56,Z 346.222,A -85,B 0,C 180,E1 -26966.351,E2 -26966.351} C_VEL
LIN {X 0,Y 134.055,Z 342.189,A -85,B 0,C 180,E1 -26968.944,E2 -26968.944} C_VEL
LIN {X 0,Y 134.079,Z 336.595,A -85,B 0,C 180,E1 -26973.011,E2 -26973.011} C_VEL
LIN {X 0,Y 133.632,Z 331.538,A -85,B 0,C 180,E1 -26977.351,E2 -26977.351} C_VEL
LIN {X 0,Y 132.484,Z 327.076,A -85,B 0,C 180,E1 -26982.722,E2 -26982.722} C_VEL
LIN {X 0,Y 131.479,Z 324.157,A -85,B 0,C 180,E1 -26987.654,E2 -26987.654} C_VEL
LIN {X 0,Y 131.152,Z 321.175,A -85,B 0,C 180,E1 -26993.847,E2 -26993.847} C_VEL
LIN {X 0,Y 131.135,Z 320.315,A -85,B 0,C 180,E1 -26996.928,E2 -26996.928} C_VEL
LIN {X 0,Y 131.134,Z 320.106,A -85,B 0,C 180,E1 -27000,E2 -27000} C_VEL
LIN {X 0,Y 131.224,Z 320.411,A -85,B 0,C 180,E1 -27003.07,E2 -27003.07} C_VEL
LIN {X 0,Y 131.321,Z 321.383,A -85,B 0,C 180,E1 -27006.144,E2 -27006.144} C_VEL
LIN {X 0,Y 131.881,Z 324.519,A -85,B 0,C 180,E1 -27012.307,E2 -27012.307} C_VEL
LIN {X 0,Y 132.348,Z 326.68,A -85,B 0,C 180,E1 -27015.397,E2 -27015.397} C_VEL
LIN {X 0,Y 133.031,Z 330.95,A -85,B 0,C 180,E1 -27020.083,E2 -27020.083} C_VEL
LIN {X 0,Y 133.444,Z 336.692,A -85,B 0,C 180,E1 -27024.918,E2 -27024.918} C_VEL
LIN {X 0,Y 133.538,Z 341.271,A -85,B 0,C 180,E1 -27028.272,E2 -27028.272} C_VEL
LIN {X 0,Y 133.25,Z 345.859,A -85,B 0,C 180,E1 -27031.265,E2 -27031.265} C_VEL
LIN {X 0,Y 131.671,Z 351.39,A -85,B 0,C 180,E1 -27034.175,E2 -27034.175} C_VEL
LIN {X 0,Y 129.292,Z 357.305,A -85,B 0,C 180,E1 -27037.177,E2 -27037.177} C_VEL
LIN {X 0,Y 126.185,Z 361.483,A -85,B 0,C 180,E1 -27038.762,E2 -27038.762} C_VEL
LIN {X 0,Y 119.057,Z 369.811,A -85,B 0,C 180,E1 -27042.448,E2 -27042.448} C_VEL
LIN {X 0,Y 111.543,Z 377.778,A -85,B 0,C 180,E1 -27047.364,E2 -27047.364} C_VEL
LIN {X 0,Y 105.011,Z 384.198,A -85,B 0,C 180,E1 -27052.962,E2 -27052.962} C_VEL
LIN {X 0,Y 98.924,Z 389.894,A -85,B 0,C 180,E1 -27060.177,E2 -27060.177} C_VEL
LIN {X 0,Y 94.356,Z 394.029,A -85,B 0,C 180,E1 -27068.135,E2 -27068.135} C_VEL
LIN {X 0,Y 91.742,Z 396.736,A -85,B 0,C 180,E1 -27076.713,E2 -27076.713} C_VEL
LIN {X 0,Y 90.798,Z 398.077,A -85,B 0,C 180,E1 -27085.56,E2 -27085.56} C_VEL
LIN {X 0,Y 90.907,Z 398.243,A -85,B 0,C 180,E1 -27090,E2 -27090} C_VEL
LIN {X 0,Y 91.074,Z 397.548,A -85,B 0,C 180,E1 -27098.878,E2 -27098.878} C_VEL
LIN {X 0,Y 92.829,Z 395.505,A -85,B 0,C 180,E1 -27107.628,E2 -27107.628} C_VEL
LIN {X 0,Y 96.458,Z 392.07,A -85,B 0,C 180,E1 -27115.923,E2 -27115.923} C_VEL
LIN {X 0,Y 101.794,Z 387.141,A -85,B 0,C 180,E1 -27123.527,E2 -27123.527} C_VEL
LIN {X 0,Y 108.605,Z 380.573,A -85,B 0,C 180,E1 -27130.324,E2 -27130.324} C_VEL
LIN {X 0,Y 115.741,Z 373.273,A -85,B 0,C 180,E1 -27135.518,E2 -27135.518} C_VEL
LIN {X 0,Y 122.559,Z 365.626,A -85,B 0,C 180,E1 -27139.447,E2 -27139.447} C_VEL
LIN {X 0,Y 128.183,Z 358.7,A -85,B 0,C 180,E1 -27142.171,E2 -27142.171} C_VEL
LIN {X 0,Y 129.167,Z 357.236,A -85,B 0,C 180,E1 -27142.75,E2 -27142.75} C_VEL
LIN {X 0,Y 132.267,Z 349.066,A -85,B 0,C 180,E1 -27146.884,E2 -27146.884} C_VEL
LIN {X 0,Y 133.276,Z 344.525,A -85,B 0,C 180,E1 -27149.403,E2 -27149.403} C_VEL
LIN {X 0,Y 133.436,Z 338.429,A -85,B 0,C 180,E1 -27153.557,E2 -27153.557} C_VEL
LIN {X 0,Y 133.014,Z 332.578,A -85,B 0,C 180,E1 -27158.294,E2 -27158.294} C_VEL
LIN {X 0,Y 132.597,Z 329.309,A -85,B 0,C 180,E1 -27161.457,E2 -27161.457} C_VEL
LIN {X 0,Y 132.168,Z 326.485,A -85,B 0,C 180,E1 -27164.581,E2 -27164.581} C_VEL
LIN {X 0,Y 131.697,Z 324.319,A -85,B 0,C 180,E1 -27167.675,E2 -27167.675} C_VEL
LIN {X 0,Y 131.132,Z 321.144,A -85,B 0,C 180,E1 -27173.847,E2 -27173.847} C_VEL
LIN {X 0,Y 130.961,Z 320.294,A -85,B 0,C 180,E1 -27176.924,E2 -27176.924} C_VEL
LIN {X 0,Y 130.884,Z 319.954,A -85,B 0,C 180,E1 -27180,E2 -27180} C_VEL
LIN {X 0,Y 130.846,Z 320.224,A -85,B 0,C 180,E1 -27183.079,E2 -27183.079} C_VEL
LIN {X 0,Y 130.945,Z 320.93,A -85,B 0,C 180,E1 -27186.162,E2 -27186.162} C_VEL
LIN {X 0,Y 131.872,Z 325.606,A -85,B 0,C 180,E1 -27195.455,E2 -27195.455} C_VEL
LIN {X 0,Y 132.852,Z 329.006,A -85,B 0,C 180,E1 -27200.112,E2 -27200.112} C_VEL
LIN {X 0,Y 133.549,Z 332.005,A -85,B 0,C 180,E1 -27203.349,E2 -27203.349} C_VEL
LIN {X 0,Y 133.935,Z 336.09,A -85,B 0,C 180,E1 -27206.869,E2 -27206.869} C_VEL
LIN {X 0,Y 133.963,Z 341.694,A -85,B 0,C 180,E1 -27210.974,E2 -27210.974} C_VEL
LIN {X 0,Y 133.532,Z 345.666,A -85,B 0,C 180,E1 -27213.546,E2 -27213.546} C_VEL
LIN {X 0,Y 133.409,Z 346.197,A -85,B 0,C 180,E1 -27213.843,E2 -27213.843} C_VEL
LIN {X 0,Y 132.384,Z 348.736,A -85,B 0,C 180,E1 -27215.025,E2 -27215.025} C_VEL
LIN {X 0,Y 129.527,Z 352.875,A -85,B 0,C 180,E1 -27216.376,E2 -27216.376} C_VEL
LIN {X 0,Y 125.76,Z 356.937,A -85,B 0,C 180,E1 -27217.395,E2 -27217.395} C_VEL
LIN {X 0,Y 119.968,Z 362.296,A -85,B 0,C 180,E1 -27218.733,E2 -27218.733} C_VEL
LIN {X 0,Y 115.903,Z 366.089,A -85,B 0,C 180,E1 -27220.122,E2 -27220.122} C_VEL
LIN {X 0,Y 114.723,Z 367.27,A -85,B 0,C 180,E1 -27220.728,E2 -27220.728} C_VEL
LIN {X 0,Y 107.323,Z 374.585,A -85,B 0,C 180,E1 -27225.255,E2 -27225.255} C_VEL
LIN {X 0,Y 100.379,Z 380.974,A -85,B 0,C 180,E1 -27230.94,E2 -27230.94} C_VEL
LIN {X 0,Y 95.262,Z 385.401,A -85,B 0,C 180,E1 -27236.406,E2 -27236.406} C_VEL
LIN {X 0,Y 90.838,Z 388.878,A -85,B 0,C 180,E1 -27242.341,E2 -27242.341} C_VEL
LIN {X 0,Y 86.736,Z 392.255,A -85,B 0,C 180,E1 -27251.089,E2 -27251.089} C_VEL
LIN {X 0,Y 84.436,Z 394.253,A -85,B 0,C 180,E1 -27260.418,E2 -27260.418} C_VEL
LIN {X 0,Y 83.841,Z 394.927,A -85,B 0,C 180,E1 -27270,E2 -27270} C_VEL
LIN {X 0,Y 84.436,Z 394.295,A -85,B 0,C 180,E1 -27279.583,E2 -27279.583} C_VEL
LIN {X 0,Y 86.724,Z 392.334,A -85,B 0,C 180,E1 -27288.915,E2 -27288.915} C_VEL
LIN {X 0,Y 90.794,Z 388.996,A -85,B 0,C 180,E1 -27297.674,E2 -27297.674} C_VEL
LIN {X 0,Y 96.823,Z 384.171,A -85,B 0,C 180,E1 -27305.5,E2 -27305.5} C_VEL
LIN {X 0,Y 104.114,Z 377.716,A -85,B 0,C 180,E1 -27312.457,E2 -27312.457} C_VEL
LIN {X 0,Y 111.739,Z 370.516,A -85,B 0,C 180,E1 -27317.65,E2 -27317.65} C_VEL
LIN {X 0,Y 120.139,Z 361.603,A -85,B 0,C 180,E1 -27322.162,E2 -27322.162} C_VEL
LIN {X 0,Y 126.117,Z 354.31,A -85,B 0,C 180,E1 -27324.932,E2 -27324.932} C_VEL
LIN {X 0,Y 127.358,Z 351.471,A -85,B 0,C 180,E1 -27326.507,E2 -27326.507} C_VEL
LIN {X 0,Y 128.407,Z 348.008,A -85,B 0,C 180,E1 -27328.67,E2 -27328.67} C_VEL
LIN {X 0,Y 129.019,Z 342.223,A -85,B 0,C 180,E1 -27333.017,E2 -27333.017} C_VEL
LIN {X 0,Y 128.978,Z 336.821,A -85,B 0,C 180,E1 -27337.871,E2 -27337.871} C_VEL
LIN {X 0,Y 128.337,Z 333.413,A -85,B 0,C 180,E1 -27342.145,E2 -27342.145} C_VEL
LIN {X 0,Y 128.069,Z 332.092,A -85,B 0,C 180,E1 -27344.074,E2 -27344.074} C_VEL
LIN {X 0,Y 127.374,Z 327.399,A -85,B 0,C 180,E1 -27353.664,E2 -27353.664} C_VEL
LIN {X 0,Y 127.448,Z 326.465,A -85,B 0,C 180,E1 -27356.839,E2 -27356.839} C_VEL
LIN {X 0,Y 127.492,Z 326.207,A -85,B 0,C 180,E1 -27360,E2 -27360} C_VEL
LIN {X 0,Y 127.551,Z 326.554,A -85,B 0,C 180,E1 -27363.158,E2 -27363.158} C_VEL
LIN {X 0,Y 127.557,Z 328.099,A -85,B 0,C 180,E1 -27367.364,E2 -27367.364} C_VEL
LIN {X 0,Y 127.935,Z 330.824,A -85,B 0,C 180,E1 -27372.693,E2 -27372.693} C_VEL
LIN {X 0,Y 128.196,Z 333.19,A -85,B 0,C 180,E1 -27375.909,E2 -27375.909} C_VEL
LIN {X 0,Y 128.485,Z 335.969,A -85,B 0,C 180,E1 -27379.159,E2 -27379.159} C_VEL
LIN {X 0,Y 128.486,Z 341.601,A -85,B 0,C 180,E1 -27384.22,E2 -27384.22} C_VEL
LIN {X 0,Y 128.235,Z 346.1,A -85,B 0,C 180,E1 -27387.714,E2 -27387.714} C_VEL
LIN {X 0,Y 127.643,Z 349.984,A -85,B 0,C 180,E1 -27390.389,E2 -27390.389} C_VEL
LIN {X 0,Y 124.751,Z 357.108,A -85,B 0,C 180,E1 -27394.288,E2 -27394.288} C_VEL
LIN {X 0,Y 124.105,Z 358.411,A -85,B 0,C 180,E1 -27394.984,E2 -27394.984} C_VEL
LIN {X 0,Y 121.85,Z 361.35,A -85,B 0,C 180,E1 -27396.148,E2 -27396.148} C_VEL
LIN {X 0,Y 114.366,Z 369.677,A -85,B 0,C 180,E1 -27399.811,E2 -27399.811} C_VEL
LIN {X 0,Y 106.397,Z 377.644,A -85,B 0,C 180,E1 -27404.758,E2 -27404.758} C_VEL
LIN {X 0,Y 99.392,Z 384.063,A -85,B 0,C 180,E1 -27410.476,E2 -27410.476} C_VEL
LIN {X 0,Y 92.795,Z 389.76,A -85,B 0,C 180,E1 -27417.983,E2 -27417.983} C_VEL
LIN {X 0,Y 87.769,Z 393.894,A -85,B 0,C 180,E1 -27426.398,E2 -27426.398} C_VEL
LIN {X 0,Y 84.809,Z 396.601,A -85,B 0,C 180,E1 -27435.604,E2 -27435.604} C_VEL
LIN {X 0,Y 83.713,Z 397.942,A -85,B 0,C 180,E1 -27445.184,E2 -27445.184} C_VEL
LIN {X 0,Y 83.805,Z 398.108,A -85,B 0,C 180,E1 -27450,E2 -27450} C_VEL
LIN {X 0,Y 84.041,Z 397.413,A -85,B 0,C 180,E1 -27459.628,E2 -27459.628} C_VEL
LIN {X 0,Y 86.049,Z 395.369,A -85,B 0,C 180,E1 -27469.068,E2 -27469.068} C_VEL
LIN {X 0,Y 90.096,Z 391.934,A -85,B 0,C 180,E1 -27477.906,E2 -27477.906} C_VEL
LIN {X 0,Y 95.9,Z 387.004,A -85,B 0,C 180,E1 -27485.893,E2 -27485.893} C_VEL
LIN {X 0,Y 103.251,Z 380.436,A -85,B 0,C 180,E1 -27492.896,E2 -27492.896} C_VEL
LIN {X 0,Y 110.837,Z 373.136,A -85,B 0,C 180,E1 -27498.163,E2 -27498.163} C_VEL
LIN {X 0,Y 119.288,Z 364.093,A -85,B 0,C 180,E1 -27502.69,E2 -27502.69} C_VEL
LIN {X 0,Y 122.973,Z 359.779,A -85,B 0,C 180,E1 -27504.355,E2 -27504.355} C_VEL
LIN {X 0,Y 123.951,Z 358.343,A -85,B 0,C 180,E1 -27504.953,E2 -27504.953} C_VEL
LIN {X 0,Y 126.813,Z 351.805,A -85,B 0,C 180,E1 -27508.479,E2 -27508.479} C_VEL
LIN {X 0,Y 127.792,Z 348.605,A -85,B 0,C 180,E1 -27510.333,E2 -27510.333} C_VEL
LIN {X 0,Y 128.319,Z 343.537,A -85,B 0,C 180,E1 -27514.014,E2 -27514.014} C_VEL
LIN {X 0,Y 128.352,Z 338.185,A -85,B 0,C 180,E1 -27518.567,E2 -27518.567} C_VEL
LIN {X 0,Y 128.192,Z 334.683,A -85,B 0,C 180,E1 -27522.102,E2 -27522.102} C_VEL
LIN {X 0,Y 127.923,Z 331.69,A -85,B 0,C 180,E1 -27525.687,E2 -27525.687} C_VEL
LIN {X 0,Y 127.457,Z 328.914,A -85,B 0,C 180,E1 -27530.479,E2 -27530.479} C_VEL
LIN {X 0,Y 127.379,Z 327.386,A -85,B 0,C 180,E1 -27533.665,E2 -27533.665} C_VEL
LIN {X 0,Y 127.295,Z 326.437,A -85,B 0,C 180,E1 -27536.835,E2 -27536.835} C_VEL
LIN {X 0,Y 127.254,Z 326.052,A -85,B 0,C 180,E1 -27540,E2 -27540} C_VEL
LIN {X 0,Y 127.181,Z 326.347,A -85,B 0,C 180,E1 -27543.168,E2 -27543.168} C_VEL
LIN {X 0,Y 127.179,Z 327.162,A -85,B 0,C 180,E1 -27546.346,E2 -27546.346} C_VEL
LIN {X 0,Y 127.38,Z 330.102,A -85,B 0,C 180,E1 -27552.75,E2 -27552.75} C_VEL
LIN {X 0,Y 128.089,Z 332.807,A -85,B 0,C 180,E1 -27557.362,E2 -27557.362} C_VEL
LIN {X 0,Y 128.819,Z 336.873,A -85,B 0,C 180,E1 -27562.452,E2 -27562.452} C_VEL
LIN {X 0,Y 128.916,Z 340.543,A -85,B 0,C 180,E1 -27565.858,E2 -27565.858} C_VEL
LIN {X 0,Y 128.53,Z 346.296,A -85,B 0,C 180,E1 -27570.384,E2 -27570.384} C_VEL
LIN {X 0,Y 127.684,Z 350.07,A -85,B 0,C 180,E1 -27572.887,E2 -27572.887} C_VEL
LIN {X 0,Y 126.118,Z 353.984,A -85,B 0,C 180,E1 -27575.101,E2 -27575.101} C_VEL
LIN {X 0,Y 118.959,Z 362.663,A -85,B 0,C 180,E1 -27578.483,E2 -27578.483} C_VEL
LIN {X 0,Y 114.723,Z 367.27,A -85,B 0,C 180,E1 -27580.728,E2 -27580.728} C_VEL
LIN {X 0,Y 111.08,Z 370.619,A -85,B 0,C 180,E1 -27582.39,E2 -27582.39} C_VEL
LIN {X 0,Y 103.787,Z 375.699,A -85,B 0,C 180,E1 -27584.747,E2 -27584.747} C_VEL
LIN {X 0,Y 96.513,Z 380.251,A -85,B 0,C 180,E1 -27587.576,E2 -27587.576} C_VEL
LIN {X 0,Y 93.03,Z 382.691,A -85,B 0,C 180,E1 -27590.011,E2 -27590.011} C_VEL
LIN {X 0,Y 87.705,Z 386.772,A -85,B 0,C 180,E1 -27595.881,E2 -27595.881} C_VEL
LIN {X 0,Y 82.083,Z 390.88,A -85,B 0,C 180,E1 -27604.653,E2 -27604.653} C_VEL
LIN {X 0,Y 78.468,Z 393.558,A -85,B 0,C 180,E1 -27614.414,E2 -27614.414} C_VEL
LIN {X 0,Y 76.884,Z 394.888,A -85,B 0,C 180,E1 -27624.756,E2 -27624.756} C_VEL
LIN {X 0,Y 76.757,Z 395.061,A -85,B 0,C 180,E1 -27630.001,E2 -27630.001} C_VEL
LIN {X 0,Y 77.448,Z 394.429,A -85,B 0,C 180,E1 -27640.457,E2 -27640.457} C_VEL
LIN {X 0,Y 80.027,Z 392.468,A -85,B 0,C 180,E1 -27650.566,E2 -27650.566} C_VEL
LIN {X 0,Y 84.551,Z 389.13,A -85,B 0,C 180,E1 -27659.917,E2 -27659.917} C_VEL
LIN {X 0,Y 91.094,Z 384.306,A -85,B 0,C 180,E1 -27668.113,E2 -27668.113} C_VEL
LIN {X 0,Y 97.127,Z 379.42,A -85,B 0,C 180,E1 -27673.79,E2 -27673.79} C_VEL
LIN {X 0,Y 104.676,Z 372.872,A -85,B 0,C 180,E1 -27679.055,E2 -27679.055} C_VEL
LIN {X 0,Y 113.333,Z 364.449,A -85,B 0,C 180,E1 -27683.723,E2 -27683.723} C_VEL
LIN {X 0,Y 120.81,Z 356.065,A -85,B 0,C 180,E1 -27687.127,E2 -27687.127} C_VEL
LIN {X 0,Y 121.669,Z 354.648,A -85,B 0,C 180,E1 -27687.851,E2 -27687.851} C_VEL
LIN {X 0,Y 122.853,Z 351.599,A -85,B 0,C 180,E1 -27689.86,E2 -27689.86} C_VEL
LIN {X 0,Y 123.785,Z 346.437,A -85,B 0,C 180,E1 -27694.066,E2 -27694.066} C_VEL
LIN {X 0,Y 124.086,Z 342.345,A -85,B 0,C 180,E1 -27698.008,E2 -27698.008} C_VEL
LIN {X 0,Y 123.859,Z 339.307,A -85,B 0,C 180,E1 -27701.815,E2 -27701.815} C_VEL
LIN {X 0,Y 123.338,Z 336.379,A -85,B 0,C 180,E1 -27706.825,E2 -27706.825} C_VEL
LIN {X 0,Y 123.276,Z 333.455,A -85,B 0,C 180,E1 -27713.453,E2 -27713.453} C_VEL
LIN {X 0,Y 123.477,Z 332.428,A -85,B 0,C 180,E1 -27716.737,E2 -27716.737} C_VEL
LIN {X 0,Y 123.576,Z 332.118,A -85,B 0,C 180,E1 -27720,E2 -27720} C_VEL
LIN {X 0,Y 123.574,Z 332.545,A -85,B 0,C 180,E1 -27723.26,E2 -27723.26} C_VEL
LIN {X 0,Y 123.494,Z 333.669,A -85,B 0,C 180,E1 -27726.535,E2 -27726.535} C_VEL
LIN {X 0,Y 123.675,Z 336.953,A -85,B 0,C 180,E1 -27733.138,E2 -27733.138} C_VEL
LIN {X 0,Y 123.776,Z 340.843,A -85,B 0,C 180,E1 -27738.197,E2 -27738.197} C_VEL
LIN {X 0,Y 123.377,Z 346.327,A -85,B 0,C 180,E1 -27743.499,E2 -27743.499} C_VEL
LIN {X 0,Y 122.722,Z 350.908,A -85,B 0,C 180,E1 -27747.267,E2 -27747.267} C_VEL
LIN {X 0,Y 122.261,Z 352.787,A -85,B 0,C 180,E1 -27748.665,E2 -27748.665} C_VEL
LIN {X 0,Y 119.744,Z 358.269,A -85,B 0,C 180,E1 -27751.885,E2 -27751.885} C_VEL
LIN {X 0,Y 119.074,Z 359.558,A -85,B 0,C 180,E1 -27752.611,E2 -27752.611} C_VEL
LIN {X 0,Y 116.455,Z 362.707,A -85,B 0,C 180,E1 -27753.92,E2 -27753.92} C_VEL
LIN {X 0,Y 108.681,Z 370.779,A -85,B 0,C 180,E1 -27757.611,E2 -27757.611} C_VEL
LIN {X 0,Y 100.356,Z 378.522,A -85,B 0,C 180,E1 -27762.664,E2 -27762.664} C_VEL
LIN {X 0,Y 93.99,Z 383.929,A -85,B 0,C 180,E1 -27767.703,E2 -27767.703} C_VEL
LIN {X 0,Y 86.825,Z 389.625,A -85,B 0,C 180,E1 -27775.485,E2 -27775.485} C_VEL
LIN {X 0,Y 81.282,Z 393.759,A -85,B 0,C 180,E1 -27784.384,E2 -27784.384} C_VEL
LIN {X 0,Y 77.923,Z 396.466,A -85,B 0,C 180,E1 -27794.301,E2 -27794.301} C_VEL
LIN {X 0,Y 76.62,Z 397.807,A -85,B 0,C 180,E1 -27804.737,E2 -27804.737} C_VEL
LIN {X 0,Y 76.702,Z 397.974,A -85,B 0,C 180,E1 -27809.999,E2 -27809.999} C_VEL
LIN {X 0,Y 77.037,Z 397.277,A -85,B 0,C 180,E1 -27820.512,E2 -27820.512} C_VEL
LIN {X 0,Y 79.319,Z 395.233,A -85,B 0,C 180,E1 -27830.757,E2 -27830.757} C_VEL
LIN {X 0,Y 83.857,Z 391.798,A -85,B 0,C 180,E1 -27840.189,E2 -27840.189} C_VEL
LIN {X 0,Y 90.198,Z 386.867,A -85,B 0,C 180,E1 -27848.56,E2 -27848.56} C_VEL
LIN {X 0,Y 98.143,Z 380.299,A -85,B 0,C 180,E1 -27855.733,E2 -27855.733} C_VEL
LIN {X 0,Y 106.202,Z 372.998,A -85,B 0,C 180,E1 -27861.038,E2 -27861.038} C_VEL
LIN {X 0,Y 115.112,Z 363.956,A -85,B 0,C 180,E1 -27865.509,E2 -27865.509} C_VEL
LIN {X 0,Y 117.778,Z 360.977,A -85,B 0,C 180,E1 -27866.658,E2 -27866.658} C_VEL
LIN {X 0,Y 118.895,Z 359.491,A -85,B 0,C 180,E1 -27867.333,E2 -27867.333} C_VEL
LIN {X 0,Y 121.435,Z 354.407,A -85,B 0,C 180,E1 -27870.241,E2 -27870.241} C_VEL
LIN {X 0,Y 122.166,Z 352.514,A -85,B 0,C 180,E1 -27871.393,E2 -27871.393} C_VEL
LIN {X 0,Y 123.011,Z 348.282,A -85,B 0,C 180,E1 -27874.63,E2 -27874.63} C_VEL
LIN {X 0,Y 123.443,Z 343.693,A -85,B 0,C 180,E1 -27878.731,E2 -27878.731} C_VEL
LIN {X 0,Y 123.618,Z 340.672,A -85,B 0,C 180,E1 -27881.779,E2 -27881.779} C_VEL
LIN {X 0,Y 123.59,Z 337.887,A -85,B 0,C 180,E1 -27885.175,E2 -27885.175} C_VEL
LIN {X 0,Y 123.315,Z 334.979,A -85,B 0,C 180,E1 -27890.156,E2 -27890.156} C_VEL
LIN {X 0,Y 123.323,Z 333.451,A -85,B 0,C 180,E1 -27893.456,E2 -27893.456} C_VEL
LIN {X 0,Y 123.329,Z 332.419,A -85,B 0,C 180,E1 -27896.733,E2 -27896.733} C_VEL
LIN {X 0,Y 123.341,Z 331.971,A -85,B 0,C 180,E1 -27900,E2 -27900} C_VEL
LIN {X 0,Y 123.228,Z 332.294,A -85,B 0,C 180,E1 -27903.27,E2 -27903.27} C_VEL
LIN {X 0,Y 123.037,Z 333.58,A -85,B 0,C 180,E1 -27907.445,E2 -27907.445} C_VEL
LIN {X 0,Y 123.258,Z 336.679,A -85,B 0,C 180,E1 -27914.231,E2 -27914.231} C_VEL
LIN {X 0,Y 123.685,Z 339.083,A -85,B 0,C 180,E1 -27918.211,E2 -27918.211} C_VEL
LIN {X 0,Y 123.951,Z 341.779,A -85,B 0,C 180,E1 -27921.711,E2 -27921.711} C_VEL
LIN {X 0,Y 123.805,Z 344.809,A -85,B 0,C 180,E1 -27924.733,E2 -27924.733} C_VEL
LIN {X 0,Y 123.346,Z 348.683,A -85,B 0,C 180,E1 -27928.103,E2 -27928.103} C_VEL
LIN {X 0,Y 122.568,Z 352.028,A -85,B 0,C 180,E1 -27930.673,E2 -27930.673} C_VEL
LIN {X 0,Y 121.628,Z 354.348,A -85,B 0,C 180,E1 -27932.174,E2 -27932.174} C_VEL
LIN {X 0,Y 120.872,Z 355.742,A -85,B 0,C 180,E1 -27932.954,E2 -27932.954} C_VEL
LIN {X 0,Y 113.382,Z 364.149,A -85,B 0,C 180,E1 -27936.312,E2 -27936.312} C_VEL
LIN {X 0,Y 104.728,Z 372.625,A -85,B 0,C 180,E1 -27940.979,E2 -27940.979} C_VEL
LIN {X 0,Y 96.68,Z 379.638,A -85,B 0,C 180,E1 -27946.63,E2 -27946.63} C_VEL
LIN {X 0,Y 93.03,Z 382.691,A -85,B 0,C 180,E1 -27950.011,E2 -27950.011} C_VEL
LIN {X 0,Y 89.669,Z 384.989,A -85,B 0,C 180,E1 -27952.688,E2 -27952.688} C_VEL
LIN {X 0,Y 82.889,Z 388.204,A -85,B 0,C 180,E1 -27956.989,E2 -27956.989} C_VEL
LIN {X 0,Y 77.641,Z 390.361,A -85,B 0,C 180,E1 -27960.989,E2 -27960.989} C_VEL
LIN {X 0,Y 74.653,Z 391.749,A -85,B 0,C 180,E1 -27964.695,E2 -27964.695} C_VEL
LIN {X 0,Y 73.973,Z 392.124,A -85,B 0,C 180,E1 -27966.085,E2 -27966.085} C_VEL
LIN {X 0,Y 71.655,Z 393.693,A -85,B 0,C 180,E1 -27972.888,E2 -27972.888} C_VEL
LIN {X 0,Y 69.814,Z 395.023,A -85,B 0,C 180,E1 -27984.223,E2 -27984.223} C_VEL
LIN {X 0,Y 69.666,Z 395.196,A -85,B 0,C 180,E1 -27990.001,E2 -27990.001} C_VEL
LIN {X 0,Y 70.471,Z 394.564,A -85,B 0,C 180,E1 -28001.506,E2 -28001.506} C_VEL
LIN {X 0,Y 73.4,Z 392.603,A -85,B 0,C 180,E1 -28012.52,E2 -28012.52} C_VEL
LIN {X 0,Y 78.463,Z 389.264,A -85,B 0,C 180,E1 -28022.509,E2 -28022.509} C_VEL
LIN {X 0,Y 85.582,Z 384.44,A -85,B 0,C 180,E1 -28031.069,E2 -28031.069} C_VEL
LIN {X 0,Y 91.901,Z 379.73,A -85,B 0,C 180,E1 -28036.689,E2 -28036.689} C_VEL
LIN {X 0,Y 100.15,Z 373.006,A -85,B 0,C 180,E1 -28042.136,E2 -28042.136} C_VEL
LIN {X 0,Y 107.925,Z 365.931,A -85,B 0,C 180,E1 -28046.128,E2 -28046.128} C_VEL
LIN {X 0,Y 115.798,Z 357.719,A -85,B 0,C 180,E1 -28049.527,E2 -28049.527} C_VEL
LIN {X 0,Y 116.631,Z 356.443,A -85,B 0,C 180,E1 -28050.204,E2 -28050.204} C_VEL
LIN {X 0,Y 117.746,Z 353.616,A -85,B 0,C 180,E1 -28052.385,E2 -28052.385} C_VEL
LIN {X 0,Y 118.526,Z 350.218,A -85,B 0,C 180,E1 -28055.476,E2 -28055.476} C_VEL
LIN {X 0,Y 119.032,Z 346.666,A -85,B 0,C 180,E1 -28059.252,E2 -28059.252} C_VEL
LIN {X 0,Y 119.025,Z 344.126,A -85,B 0,C 180,E1 -28062.828,E2 -28062.828} C_VEL
LIN {X 0,Y 118.855,Z 342.168,A -85,B 0,C 180,E1 -28066.318,E2 -28066.318} C_VEL
LIN {X 0,Y 118.897,Z 339.287,A -85,B 0,C 180,E1 -28073.21,E2 -28073.21} C_VEL
LIN {X 0,Y 119.208,Z 338.225,A -85,B 0,C 180,E1 -28076.62,E2 -28076.62} C_VEL
LIN {X 0,Y 119.377,Z 337.851,A -85,B 0,C 180,E1 -28080,E2 -28080} C_VEL
LIN {X 0,Y 119.315,Z 338.341,A -85,B 0,C 180,E1 -28083.377,E2 -28083.377} C_VEL
LIN {X 0,Y 119.133,Z 339.516,A -85,B 0,C 180,E1 -28086.776,E2 -28086.776} C_VEL
LIN {X 0,Y 119.021,Z 341.062,A -85,B 0,C 180,E1 -28090.203,E2 -28090.203} C_VEL
LIN {X 0,Y 119.018,Z 343.002,A -85,B 0,C 180,E1 -28093.662,E2 -28093.662} C_VEL
LIN {X 0,Y 118.902,Z 345.571,A -85,B 0,C 180,E1 -28097.19,E2 -28097.19} C_VEL
LIN {X 0,Y 118.089,Z 350.904,A -85,B 0,C 180,E1 -28102.758,E2 -28102.758} C_VEL
LIN {X 0,Y 117.261,Z 354.532,A -85,B 0,C 180,E1 -28105.969,E2 -28105.969} C_VEL
LIN {X 0,Y 116.703,Z 356.094,A -85,B 0,C 180,E1 -28107.171,E2 -28107.171} C_VEL
LIN {X 0,Y 113.941,Z 361.081,A -85,B 0,C 180,E1 -28110.283,E2 -28110.283} C_VEL
LIN {X 0,Y 105.791,Z 369.41,A -85,B 0,C 180,E1 -28113.858,E2 -28113.858} C_VEL
LIN {X 0,Y 96.876,Z 377.376,A -85,B 0,C 180,E1 -28118.75,E2 -28118.75} C_VEL
LIN {X 0,Y 88.829,Z 383.795,A -85,B 0,C 180,E1 -28124.596,E2 -28124.596} C_VEL
LIN {X 0,Y 81.042,Z 389.491,A -85,B 0,C 180,E1 -28132.623,E2 -28132.623} C_VEL
LIN {X 0,Y 74.918,Z 393.625,A -85,B 0,C 180,E1 -28142.027,E2 -28142.027} C_VEL
LIN {X 0,Y 71.092,Z 396.331,A -85,B 0,C 180,E1 -28152.748,E2 -28152.748} C_VEL
LIN {X 0,Y 69.546,Z 397.672,A -85,B 0,C 180,E1 -28164.199,E2 -28164.199} C_VEL
LIN {X 0,Y 69.593,Z 397.839,A -85,B 0,C 180,E1 -28169.999,E2 -28169.999} C_VEL
LIN {X 0,Y 70.041,Z 397.142,A -85,B 0,C 180,E1 -28181.576,E2 -28181.576} C_VEL
LIN {X 0,Y 72.673,Z 395.096,A -85,B 0,C 180,E1 -28192.757,E2 -28192.757} C_VEL
LIN {X 0,Y 77.755,Z 391.661,A -85,B 0,C 180,E1 -28202.841,E2 -28202.841} C_VEL
LIN {X 0,Y 84.724,Z 386.73,A -85,B 0,C 180,E1 -28211.576,E2 -28211.576} C_VEL
LIN {X 0,Y 93.285,Z 380.162,A -85,B 0,C 180,E1 -28218.885,E2 -28218.885} C_VEL
LIN {X 0,Y 101.865,Z 372.861,A -85,B 0,C 180,E1 -28224.161,E2 -28224.161} C_VEL
LIN {X 0,Y 111.238,Z 363.818,A -85,B 0,C 180,E1 -28228.532,E2 -28228.532} C_VEL
LIN {X 0,Y 113.882,Z 360.835,A -85,B 0,C 180,E1 -28229.766,E2 -28229.766} C_VEL
LIN {X 0,Y 116.336,Z 356.46,A -85,B 0,C 180,E1 -28232.452,E2 -28232.452} C_VEL
LIN {X 0,Y 117.199,Z 354.231,A -85,B 0,C 180,E1 -28234.091,E2 -28234.091} C_VEL
LIN {X 0,Y 117.989,Z 350.71,A -85,B 0,C 180,E1 -28237.222,E2 -28237.222} C_VEL
LIN {X 0,Y 118.761,Z 345.392,A -85,B 0,C 180,E1 -28242.789,E2 -28242.789} C_VEL
LIN {X 0,Y 118.917,Z 342.747,A -85,B 0,C 180,E1 -28246.326,E2 -28246.326} C_VEL
LIN {X 0,Y 118.87,Z 340.859,A -85,B 0,C 180,E1 -28249.784,E2 -28249.784} C_VEL
LIN {X 0,Y 118.972,Z 339.312,A -85,B 0,C 180,E1 -28253.215,E2 -28253.215} C_VEL
LIN {X 0,Y 119.081,Z 338.211,A -85,B 0,C 180,E1 -28256.617,E2 -28256.617} C_VEL
LIN {X 0,Y 119.151,Z 337.704,A -85,B 0,C 180,E1 -28260,E2 -28260} C_VEL
LIN {X 0,Y 118.968,Z 338.089,A -85,B 0,C 180,E1 -28263.387,E2 -28263.387} C_VEL
LIN {X 0,Y 118.692,Z 339.263,A -85,B 0,C 180,E1 -28267.35,E2 -28267.35} C_VEL
LIN {X 0,Y 118.668,Z 341.964,A -85,B 0,C 180,E1 -28273.704,E2 -28273.704} C_VEL
LIN {X 0,Y 118.881,Z 343.888,A -85,B 0,C 180,E1 -28277.193,E2 -28277.193} C_VEL
LIN {X 0,Y 118.919,Z 346.391,A -85,B 0,C 180,E1 -28280.769,E2 -28280.769} C_VEL
LIN {X 0,Y 118.445,Z 349.929,A -85,B 0,C 180,E1 -28284.542,E2 -28284.542} C_VEL
LIN {X 0,Y 117.335,Z 354.48,A -85,B 0,C 180,E1 -28288.632,E2 -28288.632} C_VEL
LIN {X 0,Y 116.584,Z 356.151,A -85,B 0,C 180,E1 -28289.822,E2 -28289.822} C_VEL
LIN {X 0,Y 115.843,Z 357.407,A -85,B 0,C 180,E1 -28290.544,E2 -28290.544} C_VEL
LIN {X 0,Y 106.665,Z 366.909,A -85,B 0,C 180,E1 -28294.553,E2 -28294.553} C_VEL
LIN {X 0,Y 97.729,Z 374.858,A -85,B 0,C 180,E1 -28299.37,E2 -28299.37} C_VEL
LIN {X 0,Y 89.737,Z 381.248,A -85,B 0,C 180,E1 -28305.182,E2 -28305.182} C_VEL
LIN {X 0,Y 81.911,Z 386.908,A -85,B 0,C 180,E1 -28313.087,E2 -28313.087} C_VEL
LIN {X 0,Y 75.69,Z 391.017,A -85,B 0,C 180,E1 -28322.338,E2 -28322.338} C_VEL
LIN {X 0,Y 73.973,Z 392.124,A -85,B 0,C 180,E1 -28326.085,E2 -28326.085} C_VEL
LIN {X 0,Y 71.797,Z 393.256,A -85,B 0,C 180,E1 -28330.304,E2 -28330.304} C_VEL
LIN {X 0,Y 67.226,Z 394.625,A -85,B 0,C 180,E1 -28337.462,E2 -28337.462} C_VEL
LIN {X 0,Y 63.992,Z 395.214,A -85,B 0,C 180,E1 -28343.842,E2 -28343.842} C_VEL
LIN {X 0,Y 62.664,Z 395.334,A -85,B 0,C 180,E1 -28349.113,E2 -28349.113} C_VEL
LIN {X 0,Y 62.546,Z 395.308,A -85,B 0,C 180,E1 -28350.932,E2 -28350.932} C_VEL
LIN {X 0,Y 63.517,Z 394.698,A -85,B 0,C 180,E1 -28362.786,E2 -28362.786} C_VEL
LIN {X 0,Y 66.862,Z 392.738,A -85,B 0,C 180,E1 -28374.864,E2 -28374.864} C_VEL
LIN {X 0,Y 72.568,Z 389.398,A -85,B 0,C 180,E1 -28385.528,E2 -28385.528} C_VEL
LIN {X 0,Y 78.299,Z 385.947,A -85,B 0,C 180,E1 -28392.314,E2 -28392.314} C_VEL
LIN {X 0,Y 85.499,Z 381.034,A -85,B 0,C 180,E1 -28398.882,E2 -28398.882} C_VEL
LIN {X 0,Y 94.627,Z 374.209,A -85,B 0,C 180,E1 -28404.784,E2 -28404.784} C_VEL
LIN {X 0,Y 104.127,Z 366.064,A -85,B 0,C 180,E1 -28409.38,E2 -28409.38} C_VEL
LIN {X 0,Y 111.187,Z 359.045,A -85,B 0,C 180,E1 -28412.243,E2 -28412.243} C_VEL
LIN {X 0,Y 111.646,Z 358.4,A -85,B 0,C 180,E1 -28412.65,E2 -28412.65} C_VEL
LIN {X 0,Y 112.696,Z 355.7,A -85,B 0,C 180,E1 -28415.105,E2 -28415.105} C_VEL
LIN {X 0,Y 113.529,Z 352.795,A -85,B 0,C 180,E1 -28418.215,E2 -28418.215} C_VEL
LIN {X 0,Y 113.987,Z 349.87,A -85,B 0,C 180,E1 -28422.044,E2 -28422.044} C_VEL
LIN {X 0,Y 113.994,Z 347.859,A -85,B 0,C 180,E1 -28425.723,E2 -28425.723} C_VEL
LIN {X 0,Y 114.228,Z 344.916,A -85,B 0,C 180,E1 -28432.931,E2 -28432.931} C_VEL
LIN {X 0,Y 114.651,Z 343.829,A -85,B 0,C 180,E1 -28436.485,E2 -28436.485} C_VEL
LIN {X 0,Y 114.917,Z 343.375,A -85,B 0,C 180,E1 -28440,E2 -28440} C_VEL
LIN {X 0,Y 114.756,Z 343.963,A -85,B 0,C 180,E1 -28443.511,E2 -28443.511} C_VEL
LIN {X 0,Y 114.467,Z 345.169,A -85,B 0,C 180,E1 -28447.053,E2 -28447.053} C_VEL
LIN {X 0,Y 114.168,Z 347.711,A -85,B 0,C 180,E1 -28452.442,E2 -28452.442} C_VEL
LIN {X 0,Y 113.901,Z 350.108,A -85,B 0,C 180,E1 -28456.121,E2 -28456.121} C_VEL
LIN {X 0,Y 112.882,Z 354.327,A -85,B 0,C 180,E1 -28460.948,E2 -28460.948} C_VEL
LIN {X 0,Y 111.9,Z 357.502,A -85,B 0,C 180,E1 -28464.094,E2 -28464.094} C_VEL
LIN {X 0,Y 110.902,Z 359.69,A -85,B 0,C 180,E1 -28465.821,E2 -28465.821} C_VEL
LIN {X 0,Y 108.694,Z 362.885,A -85,B 0,C 180,E1 -28467.841,E2 -28467.841} C_VEL
LIN {X 0,Y 99.216,Z 371.746,A -85,B 0,C 180,E1 -28471.785,E2 -28471.785} C_VEL
LIN {X 0,Y 91.28,Z 378.254,A -85,B 0,C 180,E1 -28476.056,E2 -28476.056} C_VEL
LIN {X 0,Y 83.953,Z 383.66,A -85,B 0,C 180,E1 -28481.111,E2 -28481.111} C_VEL
LIN {X 0,Y 75.491,Z 389.356,A -85,B 0,C 180,E1 -28489.33,E2 -28489.33} C_VEL
LIN {X 0,Y 68.708,Z 393.49,A -85,B 0,C 180,E1 -28499.239,E2 -28499.239} C_VEL
LIN {X 0,Y 64.295,Z 396.196,A -85,B 0,C 180,E1 -28510.856,E2 -28510.856} C_VEL
LIN {X 0,Y 62.493,Z 397.538,A -85,B 0,C 180,E1 -28523.542,E2 -28523.542} C_VEL
LIN {X 0,Y 62.504,Z 397.704,A -85,B 0,C 180,E1 -28529.999,E2 -28529.999} C_VEL
LIN {X 0,Y 63.087,Z 397.007,A -85,B 0,C 180,E1 -28542.873,E2 -28542.873} C_VEL
LIN {X 0,Y 66.136,Z 394.96,A -85,B 0,C 180,E1 -28555.154,E2 -28555.154} C_VEL
LIN {X 0,Y 71.839,Z 391.525,A -85,B 0,C 180,E1 -28565.942,E2 -28565.942} C_VEL
LIN {X 0,Y 79.512,Z 386.593,A -85,B 0,C 180,E1 -28575,E2 -28575} C_VEL
LIN {X 0,Y 88.747,Z 380.025,A -85,B 0,C 180,E1 -28582.364,E2 -28582.364} C_VEL
LIN {X 0,Y 97.847,Z 372.723,A -85,B 0,C 180,E1 -28587.56,E2 -28587.56} C_VEL
LIN {X 0,Y 107.696,Z 363.681,A -85,B 0,C 180,E1 -28591.761,E2 -28591.761} C_VEL
LIN {X 0,Y 109.342,Z 361.719,A -85,B 0,C 180,E1 -28592.719,E2 -28592.719} C_VEL
LIN {X 0,Y 111.103,Z 358.997,A -85,B 0,C 180,E1 -28594.501,E2 -28594.501} C_VEL
LIN {X 0,Y 112.204,Z 356.174,A -85,B 0,C 180,E1 -28596.954,E2 -28596.954} C_VEL
LIN {X 0,Y 113.098,Z 352.736,A -85,B 0,C 180,E1 -28600.538,E2 -28600.538} C_VEL
LIN {X 0,Y 113.75,Z 349.948,A -85,B 0,C 180,E1 -28603.858,E2 -28603.858} C_VEL
LIN {X 0,Y 114.063,Z 347.478,A -85,B 0,C 180,E1 -28607.546,E2 -28607.546} C_VEL
LIN {X 0,Y 114.327,Z 344.964,A -85,B 0,C 180,E1 -28612.938,E2 -28612.938} C_VEL
LIN {X 0,Y 114.558,Z 343.801,A -85,B 0,C 180,E1 -28616.483,E2 -28616.483} C_VEL
LIN {X 0,Y 114.683,Z 343.251,A -85,B 0,C 180,E1 -28620,E2 -28620} C_VEL
LIN {X 0,Y 114.431,Z 343.682,A -85,B 0,C 180,E1 -28623.521,E2 -28623.521} C_VEL
LIN {X 0,Y 113.922,Z 345.46,A -85,B 0,C 180,E1 -28629.226,E2 -28629.226} C_VEL
LIN {X 0,Y 113.829,Z 347.65,A -85,B 0,C 180,E1 -28634.298,E2 -28634.298} C_VEL
LIN {X 0,Y 113.859,Z 349.638,A -85,B 0,C 180,E1 -28637.977,E2 -28637.977} C_VEL
LIN {X 0,Y 113.766,Z 350.89,A -85,B 0,C 180,E1 -28639.862,E2 -28639.862} C_VEL
LIN {X 0,Y 112.925,Z 354.42,A -85,B 0,C 180,E1 -28643.862,E2 -28643.862} C_VEL
LIN {X 0,Y 112.028,Z 357.227,A -85,B 0,C 180,E1 -28646.629,E2 -28646.629} C_VEL
LIN {X 0,Y 111.251,Z 358.725,A -85,B 0,C 180,E1 -28647.821,E2 -28647.821} C_VEL
LIN {X 0,Y 102.8,Z 367.046,A -85,B 0,C 180,E1 -28651.288,E2 -28651.288} C_VEL
LIN {X 0,Y 93.368,Z 374.995,A -85,B 0,C 180,E1 -28655.985,E2 -28655.985} C_VEL
LIN {X 0,Y 84.808,Z 381.385,A -85,B 0,C 180,E1 -28661.77,E2 -28661.77} C_VEL
LIN {X 0,Y 76.342,Z 387.044,A -85,B 0,C 180,E1 -28669.878,E2 -28669.878} C_VEL
LIN {X 0,Y 69.446,Z 391.153,A -85,B 0,C 180,E1 -28679.602,E2 -28679.602} C_VEL
LIN {X 0,Y 64.88,Z 393.829,A -85,B 0,C 180,E1 -28691.037,E2 -28691.037} C_VEL
LIN {X 0,Y 62.767,Z 395.158,A -85,B 0,C 180,E1 -28703.572,E2 -28703.572} C_VEL
LIN {X 0,Y 62.546,Z 395.308,A -85,B 0,C 180,E1 -28710.932,E2 -28710.932} C_VEL
LIN {X 0,Y 62.031,Z 395.2,A -85,B 0,C 180,E1 -28716.342,E2 -28716.342} C_VEL
LIN {X 0,Y 60.392,Z 394.535,A -85,B 0,C 180,E1 -28725.495,E2 -28725.495} C_VEL
LIN {X 0,Y 59.909,Z 393.632,A -85,B 0,C 180,E1 -28733.059,E2 -28733.059} C_VEL
LIN {X 0,Y 60.902,Z 392.667,A -85,B 0,C 180,E1 -28738.555,E2 -28738.555} C_VEL
LIN {X 0,Y 61.587,Z 392.252,A -85,B 0,C 180,E1 -28740.259,E2 -28740.259} C_VEL
LIN {X 0,Y 68.914,Z 388.475,A -85,B 0,C 180,E1 -28751.521,E2 -28751.521} C_VEL
LIN {X 0,Y 77.766,Z 383.289,A -85,B 0,C 180,E1 -28760.191,E2 -28760.191} C_VEL
LIN {X 0,Y 85.283,Z 378.251,A -85,B 0,C 180,E1 -28765.496,E2 -28765.496} C_VEL
LIN {X 0,Y 94.944,Z 371.048,A -85,B 0,C 180,E1 -28770.433,E2 -28770.433} C_VEL
LIN {X 0,Y 105.093,Z 362.135,A -85,B 0,C 180,E1 -28774.53,E2 -28774.53} C_VEL
LIN {X 0,Y 106.656,Z 360.44,A -85,B 0,C 180,E1 -28775.304,E2 -28775.304} C_VEL
LIN {X 0,Y 107.841,Z 357.634,A -85,B 0,C 180,E1 -28778.436,E2 -28778.436} C_VEL
LIN {X 0,Y 108.509,Z 355.525,A -85,B 0,C 180,E1 -28781.104,E2 -28781.104} C_VEL
LIN {X 0,Y 108.894,Z 353.277,A -85,B 0,C 180,E1 -28785.039,E2 -28785.039} C_VEL
LIN {X 0,Y 109.297,Z 350.307,A -85,B 0,C 180,E1 -28792.611,E2 -28792.611} C_VEL
LIN {X 0,Y 109.802,Z 349.229,A -85,B 0,C 180,E1 -28796.33,E2 -28796.33} C_VEL
LIN {X 0,Y 110.179,Z 348.707,A -85,B 0,C 180,E1 -28800,E2 -28800} C_VEL
LIN {X 0,Y 109.927,Z 349.358,A -85,B 0,C 180,E1 -28803.665,E2 -28803.665} C_VEL
LIN {X 0,Y 109.508,Z 350.614,A -85,B 0,C 180,E1 -28807.374,E2 -28807.374} C_VEL
LIN {X 0,Y 109.191,Z 352.23,A -85,B 0,C 180,E1 -28811.133,E2 -28811.133} C_VEL
LIN {X 0,Y 108.745,Z 354.474,A -85,B 0,C 180,E1 -28814.982,E2 -28814.982} C_VEL
LIN {X 0,Y 107.135,Z 359.169,A -85,B 0,C 180,E1 -28820.737,E2 -28820.737} C_VEL
LIN {X 0,Y 105.775,Z 361.968,A -85,B 0,C 180,E1 -28823.494,E2 -28823.494} C_VEL
LIN {X 0,Y 104.062,Z 364.217,A -85,B 0,C 180,E1 -28824.944,E2 -28824.944} C_VEL
LIN {X 0,Y 94.219,Z 372.775,A -85,B 0,C 180,E1 -28828.78,E2 -28828.78} C_VEL
LIN {X 0,Y 84.587,Z 380.041,A -85,B 0,C 180,E1 -28833.811,E2 -28833.811} C_VEL
LIN {X 0,Y 74.613,Z 386.577,A -85,B 0,C 180,E1 -28841.101,E2 -28841.101} C_VEL
LIN {X 0,Y 66.189,Z 391.474,A -85,B 0,C 180,E1 -28850.425,E2 -28850.425} C_VEL
LIN {X 0,Y 59.747,Z 394.88,A -85,B 0,C 180,E1 -28861.931,E2 -28861.931} C_VEL
LIN {X 0,Y 56.152,Z 396.901,A -85,B 0,C 180,E1 -28875.503,E2 -28875.503} C_VEL
LIN {X 0,Y 55.401,Z 397.569,A -85,B 0,C 180,E1 -28889.999,E2 -28889.999} C_VEL
LIN {X 0,Y 56.149,Z 396.871,A -85,B 0,C 180,E1 -28904.496,E2 -28904.496} C_VEL
LIN {X 0,Y 59.743,Z 394.824,A -85,B 0,C 180,E1 -28918.069,E2 -28918.069} C_VEL
LIN {X 0,Y 66.174,Z 391.388,A -85,B 0,C 180,E1 -28929.585,E2 -28929.585} C_VEL
LIN {X 0,Y 74.631,Z 386.457,A -85,B 0,C 180,E1 -28938.882,E2 -28938.882} C_VEL
LIN {X 0,Y 84.581,Z 379.888,A -85,B 0,C 180,E1 -28946.193,E2 -28946.193} C_VEL
LIN {X 0,Y 94.212,Z 372.586,A -85,B 0,C 180,E1 -28951.225,E2 -28951.225} C_VEL
LIN {X 0,Y 103.953,Z 364.043,A -85,B 0,C 180,E1 -28955.076,E2 -28955.076} C_VEL
LIN {X 0,Y 105.665,Z 361.814,A -85,B 0,C 180,E1 -28956.48,E2 -28956.48} C_VEL
LIN {X 0,Y 106.414,Z 360.51,A -85,B 0,C 180,E1 -28957.61,E2 -28957.61} C_VEL
LIN {X 0,Y 107.542,Z 357.495,A -85,B 0,C 180,E1 -28960.928,E2 -28960.928} C_VEL
LIN {X 0,Y 108.727,Z 353.755,A -85,B 0,C 180,E1 -28965.833,E2 -28965.833} C_VEL
LIN {X 0,Y 109.083,Z 352.019,A -85,B 0,C 180,E1 -28968.856,E2 -28968.856} C_VEL
LIN {X 0,Y 109.394,Z 350.402,A -85,B 0,C 180,E1 -28972.618,E2 -28972.618} C_VEL
LIN {X 0,Y 109.743,Z 349.201,A -85,B 0,C 180,E1 -28976.329,E2 -28976.329} C_VEL
LIN {X 0,Y 109.954,Z 348.584,A -85,B 0,C 180,E1 -28980,E2 -28980} C_VEL
LIN {X 0,Y 109.61,Z 349.072,A -85,B 0,C 180,E1 -28983.677,E2 -28983.677} C_VEL
LIN {X 0,Y 109.171,Z 350.085,A -85,B 0,C 180,E1 -28987.398,E2 -28987.398} C_VEL
LIN {X 0,Y 108.683,Z 353.136,A -85,B 0,C 180,E1 -28994.991,E2 -28994.991} C_VEL
LIN {X 0,Y 108.464,Z 355.233,A -85,B 0,C 180,E1 -28998.904,E2 -28998.904} C_VEL
LIN {X 0,Y 107.184,Z 358.907,A -85,B 0,C 180,E1 -29003.369,E2 -29003.369} C_VEL
LIN {X 0,Y 106.62,Z 360.193,A -85,B 0,C 180,E1 -29004.757,E2 -29004.757} C_VEL
LIN {X 0,Y 103.686,Z 363.211,A -85,B 0,C 180,E1 -29006.091,E2 -29006.091} C_VEL
